  MoveL 8647 to (-40.61, 49.48, 125.68) mm, rotated rx 180 ry 0 rz 180 deg; joints [-136.108, -46.338, -97.928, 49.844, 65.111, -26.51]
  MoveL 8648 to (-40.61, 49.48, 125.68) mm, rotated rx 180 ry 0 rz 180 deg; joints [-136.108, -46.338, -97.928, 49.844, 65.111, -26.51]
  Call Extruder(456.97214)
  MoveL 8649 to (-40.56, 49.18, 125.68) mm, rotated rx 180 ry 0 rz -180 deg; joints [-136.149, -46.327, -97.959, 49.797, 65.104, -26.477]
  MoveL 8650 to (-40.56, 49.18, 125.68) mm, rotated rx 180 ry 0 rz -180 deg; joints [-136.149, -46.327, -97.959, 49.797, 65.104, -26.477]
  Call Extruder(457.10606)
  MoveL 8651 to (-40.52, 48.93, 125.68) mm, rotated rx 180 ry 0 rz 180 deg; joints [-136.184, -46.317, -97.983, 49.757, 65.098, -26.45]
  MoveL 8652 to (-40.52, 48.93, 125.68) mm, rotated rx 180 ry 0 rz 180 deg; joints [-136.184, -46.317, -97.983, 49.757, 65.098, -26.45]
  Call Extruder(457.24060)
  MoveL 8653 to (-40.47, 48.68, 125.68) mm, rotated rx 180 ry 0 rz -180 deg; joints [-136.219, -46.308, -98.006, 49.717, 65.092, -26.424]
  MoveL 8654 to (-40.47, 48.68, 125.68) mm, rotated rx 180 ry 0 rz -180 deg; joints [-136.219, -46.308, -98.006, 49.717, 65.092, -26.424]
  Call Extruder(457.37574)
  MoveL 8655 to (-40.42, 48.43, 125.68) mm, rotated rx 180 ry 0 rz 180 deg; joints [-136.254, -46.3, -98.03, 49.678, 65.086, -26.397]
  MoveL 8656 to (-40.42, 48.43, 125.68) mm, rotated rx 180 ry 0 rz 180 deg; joints [-136.254, -46.3, -98.03, 49.678, 65.086, -26.397]
  Call Extruder(457.51150)
  MoveL 8657 to (-40.37, 48.18, 125.68) mm, rotated rx 180 ry 0 rz 180 deg; joints [-136.288, -46.291, -98.053, 49.638, 65.08, -26.37]
  MoveL 8658 to (-40.37, 48.18, 125.68) mm, rotated rx 180 ry 0 rz 180 deg; joints [-136.288, -46.291, -98.053, 49.638, 65.08, -26.37]
  Call Extruder(457.64786)
  MoveL 8659 to (-40.32, 47.93, 125.68) mm, rotated rx 180 ry 0 rz 180 deg; joints [-136.323, -46.282, -98.077, 49.599, 65.074, -26.344]
  MoveL 8660 to (-40.32, 47.93, 125.68) mm, rotated rx 180 ry 0 rz 180 deg; joints [-136.323, -46.282, -98.077, 49.599, 65.074, -26.344]
  Call Extruder(457.78484)
  MoveL 8661 to (-40.27, 47.68, 125.68) mm, rotated rx 180 ry 0 rz 180 deg; joints [-136.358, -46.273, -98.1, 49.559, 65.068, -26.317]
  MoveL 8662 to (-40.27, 47.68, 125.68) mm, rotated rx 180 ry 0 rz 180 deg; joints [-136.358, -46.273, -98.1, 49.559, 65.068, -26.317]
  Call Extruder(457.92243)
  MoveL 8663 to (-40.22, 47.43, 125.68) mm, rotated rx 180 ry 0 rz 180 deg; joints [-136.393, -46.264, -98.123, 49.519, 65.062, -26.29]
  MoveL 8664 to (-40.22, 47.43, 125.68) mm, rotated rx 180 ry 0 rz 180 deg; joints [-136.393, -46.264, -98.123, 49.519, 65.062, -26.29]
  Call Extruder(458.03615)
  MoveL 8665 to (-40.17, 47.23, 125.68) mm, rotated rx -180 ry 0 rz -180 deg; joints [-136.422, -46.257, -98.142, 49.486, 65.056, -26.268]
  MoveL 8666 to (-40.17, 47.23, 125.68) mm, rotated rx -180 ry 0 rz -180 deg; joints [-136.422, -46.257, -98.142, 49.486, 65.056, -26.268]
  Call Extruder(458.15034)
  MoveL 8667 to (-40.13, 47.02, 125.68) mm, rotated rx 180 ry 0 rz 180 deg; joints [-136.452, -46.249, -98.161, 49.453, 65.051, -26.246]
  MoveL 8668 to (-40.13, 47.02, 125.68) mm, rotated rx 180 ry 0 rz 180 deg; joints [-136.452, -46.249, -98.161, 49.453, 65.051, -26.246]
  Call Extruder(458.26497)
  MoveL 8669 to (-40.08, 46.82, 125.68) mm, rotated rx 180 ry 0 rz 180 deg; joints [-136.481, -46.242, -98.18, 49.42, 65.046, -26.224]
  MoveL 8670 to (-40.08, 46.82, 125.68) mm, rotated rx 180 ry 0 rz 180 deg; joints [-136.481, -46.242, -98.18, 49.42, 65.046, -26.224]
  Call Extruder(458.38006)
  MoveL 8671 to (-40.04, 46.61, 125.68) mm, rotated rx 180 ry 0 rz -180 deg; joints [-136.51, -46.235, -98.198, 49.387, 65.04, -26.203]
  MoveL 8672 to (-40.04, 46.61, 125.68) mm, rotated rx 180 ry 0 rz -180 deg; joints [-136.51, -46.235, -98.198, 49.387, 65.04, -26.203]
  Call Extruder(458.50230)
  MoveL 8673 to (-39.98, 46.4, 125.68) mm, rotated rx 180 ry 0 rz -180 deg; joints [-136.542, -46.228, -98.217, 49.352, 65.034, -26.18]
  MoveL 8674 to (-39.98, 46.4, 125.68) mm, rotated rx 180 ry 0 rz -180 deg; joints [-136.542, -46.228, -98.217, 49.352, 65.034, -26.18]
  Call Extruder(458.63196)
  MoveL 8675 to (-39.92, 46.18, 125.68) mm, rotated rx 180 ry 0 rz -180 deg; joints [-136.576, -46.221, -98.235, 49.314, 65.026, -26.156]
  MoveL 8676 to (-39.92, 46.18, 125.68) mm, rotated rx 180 ry 0 rz -180 deg; joints [-136.576, -46.221, -98.235, 49.314, 65.026, -26.156]
  Call Extruder(458.76219)
  MoveL 8677 to (-39.85, 45.95, 125.68) mm, rotated rx -180 ry 0 rz -180 deg; joints [-136.61, -46.214, -98.253, 49.277, 65.018, -26.133]
  MoveL 8678 to (-39.85, 45.95, 125.68) mm, rotated rx -180 ry 0 rz -180 deg; joints [-136.61, -46.214, -98.253, 49.277, 65.018, -26.133]
  Call Extruder(458.89299)
  MoveL 8679 to (-39.78, 45.73, 125.68) mm, rotated rx -180 ry 0 rz 180 deg; joints [-136.644, -46.208, -98.271, 49.239, 65.01, -26.109]
  MoveL 8680 to (-39.78, 45.73, 125.68) mm, rotated rx -180 ry 0 rz 180 deg; joints [-136.644, -46.208, -98.271, 49.239, 65.01, -26.109]
  Call Extruder(459.02435)
  MoveL 8681 to (-39.71, 45.51, 125.68) mm, rotated rx 180 ry 0 rz 180 deg; joints [-136.678, -46.201, -98.289, 49.201, 65.002, -26.085]
  MoveL 8682 to (-39.71, 45.51, 125.68) mm, rotated rx 180 ry 0 rz 180 deg; joints [-136.678, -46.201, -98.289, 49.201, 65.002, -26.085]
  Call Extruder(459.13625)
  MoveL 8683 to (-39.65, 45.32, 125.68) mm, rotated rx 180 ry 0 rz -180 deg; joints [-136.707, -46.195, -98.303, 49.169, 64.996, -26.066]
  MoveL 8684 to (-39.65, 45.32, 125.68) mm, rotated rx 180 ry 0 rz -180 deg; joints [-136.707, -46.195, -98.303, 49.169, 64.996, -26.066]
  Call Extruder(459.24859)
  MoveL 8685 to (-39.59, 45.13, 125.68) mm, rotated rx -180 ry 0 rz 180 deg; joints [-136.737, -46.19, -98.318, 49.137, 64.989, -26.046]
  MoveL 8686 to (-39.59, 45.13, 125.68) mm, rotated rx -180 ry 0 rz 180 deg; joints [-136.737, -46.19, -98.318, 49.137, 64.989, -26.046]
  Call Extruder(459.36138)
  MoveL 8687 to (-39.53, 44.94, 125.68) mm, rotated rx 180 ry 0 rz 180 deg; joints [-136.766, -46.184, -98.332, 49.104, 64.982, -26.026]
  MoveL 8688 to (-39.53, 44.94, 125.68) mm, rotated rx 180 ry 0 rz 180 deg; joints [-136.766, -46.184, -98.332, 49.104, 64.982, -26.026]
  Call Extruder(459.47461)
  MoveL 8689 to (-39.47, 44.75, 125.68) mm, rotated rx 180 ry 0 rz -180 deg; joints [-136.796, -46.179, -98.347, 49.072, 64.975, -26.006]
  MoveL 8690 to (-39.47, 44.75, 125.68) mm, rotated rx 180 ry 0 rz -180 deg; joints [-136.796, -46.179, -98.347, 49.072, 64.975, -26.006]
  Call Extruder(459.58829)
  MoveL 8691 to (-39.41, 44.56, 125.68) mm, rotated rx -180 ry 0 rz 180 deg; joints [-136.825, -46.173, -98.361, 49.04, 64.968, -25.986]
  MoveL 8692 to (-39.41, 44.56, 125.68) mm, rotated rx -180 ry 0 rz 180 deg; joints [-136.825, -46.173, -98.361, 49.04, 64.968, -25.986]
  Call Extruder(459.77026)
  MoveL 8693 to (-39.29, 44.27, 125.68) mm, rotated rx 180 ry 0 rz -180 deg; joints [-136.873, -46.166, -98.381, 48.988, 64.954, -25.956]
  MoveL 8694 to (-39.29, 44.27, 125.68) mm, rotated rx 180 ry 0 rz -180 deg; joints [-136.873, -46.166, -98.381, 48.988, 64.954, -25.956]
  Call Extruder(459.95298)
  MoveL 8695 to (-39.17, 43.98, 125.68) mm, rotated rx 180 ry 0 rz -180 deg; joints [-136.922, -46.158, -98.4, 48.935, 64.941, -25.926]
  MoveL 8696 to (-39.17, 43.98, 125.68) mm, rotated rx 180 ry 0 rz -180 deg; joints [-136.922, -46.158, -98.4, 48.935, 64.941, -25.926]
  Call Extruder(460.12339)
  MoveL 8697 to (-39.05, 43.71, 125.68) mm, rotated rx 180 ry 0 rz 180 deg; joints [-136.967, -46.152, -98.417, 48.887, 64.928, -25.898]
  MoveL 8698 to (-39.05, 43.71, 125.68) mm, rotated rx 180 ry 0 rz 180 deg; joints [-136.967, -46.152, -98.417, 48.887, 64.928, -25.898]
  Call Extruder(460.28137)
  MoveL 8699 to (-38.94, 43.46, 125.68) mm, rotated rx 180 ry 0 rz 180 deg; joints [-137.009, -46.146, -98.433, 48.842, 64.916, -25.872]
  MoveL 8700 to (-38.94, 43.46, 125.68) mm, rotated rx 180 ry 0 rz 180 deg; joints [-137.009, -46.146, -98.433, 48.842, 64.916, -25.872]
  Call Extruder(460.43996)
  MoveL 8701 to (-38.84, 43.21, 125.68) mm, rotated rx -180 ry 0 rz 180 deg; joints [-137.05, -46.14, -98.449, 48.797, 64.905, -25.846]
  MoveL 8702 to (-38.84, 43.21, 125.68) mm, rotated rx -180 ry 0 rz 180 deg; joints [-137.05, -46.14, -98.449, 48.797, 64.905, -25.846]
  Call Extruder(460.64612)
  MoveL 8703 to (-38.66, 42.91, 125.68) mm, rotated rx -180 ry 0 rz -180 deg; joints [-137.107, -46.135, -98.462, 48.738, 64.886, -25.816]
  MoveL 8704 to (-38.66, 42.91, 125.68) mm, rotated rx -180 ry 0 rz -180 deg; joints [-137.107, -46.135, -98.462, 48.738, 64.886, -25.816]
  Call Extruder(460.85306)
  MoveL 8705 to (-38.49, 42.6, 125.68) mm, rotated rx -180 ry 0 rz -180 deg; joints [-137.163, -46.13, -98.476, 48.679, 64.867, -25.785]
  MoveL 8706 to (-38.49, 42.6, 125.68) mm, rotated rx -180 ry 0 rz -180 deg; joints [-137.163, -46.13, -98.476, 48.679, 64.867, -25.785]
  Call Extruder(461.06079)
  MoveL 8707 to (-38.31, 42.3, 125.68) mm, rotated rx 180 ry 0 rz 180 deg; joints [-137.219, -46.125, -98.489, 48.62, 64.848, -25.755]
  MoveL 8708 to (-38.31, 42.3, 125.68) mm, rotated rx 180 ry 0 rz 180 deg; joints [-137.219, -46.125, -98.489, 48.62, 64.848, -25.755]
  Call Extruder(461.26929)
  MoveL 8709 to (-38.13, 41.99, 125.68) mm, rotated rx 180 ry 0 rz -180 deg; joints [-137.275, -46.119, -98.502, 48.562, 64.829, -25.724]
  MoveL 8710 to (-38.13, 41.99, 125.68) mm, rotated rx 180 ry 0 rz -180 deg; joints [-137.275, -46.119, -98.502, 48.562, 64.829, -25.724]
  Call Extruder(461.44884)
  MoveL 8711 to (-37.96, 41.75, 125.68) mm, rotated rx 180 ry 0 rz 180 deg; joints [-137.324, -46.117, -98.509, 48.511, 64.81, -25.7]
  MoveL 8712 to (-37.96, 41.75, 125.68) mm, rotated rx 180 ry 0 rz 180 deg; joints [-137.324, -46.117, -98.509, 48.511, 64.81, -25.7]
  Call Extruder(461.78228)
  MoveL 8713 to (-37.63, 41.3, 125.68) mm, rotated rx 180 ry 0 rz -180 deg; joints [-137.415, -46.113, -98.52, 48.418, 64.775, -25.656]
  MoveL 8714 to (-37.63, 41.3, 125.68) mm, rotated rx 180 ry 0 rz -180 deg; joints [-137.415, -46.113, -98.52, 48.418, 64.775, -25.656]
  Call Extruder(462.11690)
  MoveL 8715 to (-37.3, 40.85, 125.68) mm, rotated rx 180 ry 0 rz 180 deg; joints [-137.506, -46.109, -98.531, 48.325, 64.74, -25.611]
  Call Extruder(462.94483)
  MoveL 8716 to (-36.39, 39.81, 125.68) mm, rotated rx 180 ry 0 rz -180 deg; joints [-137.733, -46.107, -98.535, 48.098, 64.644, -25.512]
  Call Extruder(463.77274)
  MoveL 8717 to (-35.35, 38.9, 125.68) mm, rotated rx 180 ry 0 rz -180 deg; joints [-137.958, -46.117, -98.508, 47.879, 64.536, -25.43]
  Call Extruder(463.94004)
  MoveL 8718 to (-35.13, 38.73, 125.68) mm, rotated rx 180 ry 0 rz 180 deg; joints [-138.003, -46.121, -98.498, 47.836, 64.513, -25.415]
  MoveL 8719 to (-35.13, 38.73, 125.68) mm, rotated rx 180 ry 0 rz 180 deg; joints [-138.003, -46.121, -98.498, 47.836, 64.513, -25.415]
  Call Extruder(464.27347)
  MoveL 8720 to (-34.68, 38.4, 125.68) mm, rotated rx -180 ry 0 rz 180 deg; joints [-138.092, -46.129, -98.478, 47.751, 64.466, -25.387]
  MoveL 8721 to (-34.68, 38.4, 125.68) mm, rotated rx -180 ry 0 rz 180 deg; joints [-138.092, -46.129, -98.478, 47.751, 64.466, -25.387]
  Call Extruder(464.60571)
  MoveL 8722 to (-34.23, 38.08, 125.68) mm, rotated rx -180 ry 0 rz -180 deg; joints [-138.182, -46.136, -98.458, 47.666, 64.419, -25.358]
  MoveL 8723 to (-34.23, 38.08, 125.68) mm, rotated rx -180 ry 0 rz -180 deg; joints [-138.182, -46.136, -98.458, 47.666, 64.419, -25.358]
  Call Extruder(464.72342)
  MoveL 8724 to (-34.05, 37.98, 125.68) mm, rotated rx 180 ry 0 rz -180 deg; joints [-138.213, -46.14, -98.447, 47.637, 64.402, -25.351]
  MoveL 8725 to (-34.05, 37.98, 125.68) mm, rotated rx 180 ry 0 rz -180 deg; joints [-138.213, -46.14, -98.447, 47.637, 64.402, -25.351]
  Call Extruder(464.93114)
  MoveL 8726 to (-33.75, 37.8, 125.68) mm, rotated rx 180 ry 0 rz 180 deg; joints [-138.267, -46.147, -98.429, 47.586, 64.371, -25.336]
  MoveL 8727 to (-33.75, 37.8, 125.68) mm, rotated rx 180 ry 0 rz 180 deg; joints [-138.267, -46.147, -98.429, 47.586, 64.371, -25.336]
  Call Extruder(465.13808)
  MoveL 8728 to (-33.45, 37.63, 125.68) mm, rotated rx -180 ry 0 rz 180 deg; joints [-138.322, -46.155, -98.41, 47.536, 64.339, -25.322]
  MoveL 8729 to (-33.45, 37.63, 125.68) mm, rotated rx -180 ry 0 rz 180 deg; joints [-138.322, -46.155, -98.41, 47.536, 64.339, -25.322]
  Call Extruder(465.34424)
  MoveL 8730 to (-33.14, 37.45, 125.68) mm, rotated rx 180 ry 0 rz -180 deg; joints [-138.376, -46.162, -98.39, 47.485, 64.308, -25.308]
  MoveL 8731 to (-33.14, 37.45, 125.68) mm, rotated rx 180 ry 0 rz -180 deg; joints [-138.376, -46.162, -98.39, 47.485, 64.308, -25.308]
  Call Extruder(465.52591)
  MoveL 8732 to (-32.87, 37.31, 125.68) mm, rotated rx -180 ry 0 rz -180 deg; joints [-138.424, -46.169, -98.371, 47.442, 64.28, -25.298]
  MoveL 8733 to (-32.87, 37.31, 125.68) mm, rotated rx -180 ry 0 rz -180 deg; joints [-138.424, -46.169, -98.371, 47.442, 64.28, -25.298]
  Call Extruder(465.68390)
  MoveL 8734 to (-32.62, 37.2, 125.68) mm, rotated rx 180 ry 0 rz -180 deg; joints [-138.464, -46.177, -98.351, 47.406, 64.254, -25.29]
  MoveL 8735 to (-32.62, 37.2, 125.68) mm, rotated rx 180 ry 0 rz -180 deg; joints [-138.464, -46.177, -98.351, 47.406, 64.254, -25.29]
  Call Extruder(465.84129)
  MoveL 8736 to (-32.37, 37.09, 125.68) mm, rotated rx -180 ry 0 rz -180 deg; joints [-138.504, -46.184, -98.331, 47.37, 64.229, -25.283]
  MoveL 8737 to (-32.37, 37.09, 125.68) mm, rotated rx -180 ry 0 rz -180 deg; joints [-138.504, -46.184, -98.331, 47.37, 64.229, -25.283]
  Call Extruder(465.98171)
  MoveL 8738 to (-32.14, 37, 125.68) mm, rotated rx -180 ry 0 rz -180 deg; joints [-138.54, -46.191, -98.313, 47.339, 64.206, -25.276]
  MoveL 8739 to (-32.14, 37, 125.68) mm, rotated rx -180 ry 0 rz -180 deg; joints [-138.54, -46.191, -98.313, 47.339, 64.206, -25.276]
  Call Extruder(466.13359)
  MoveL 8740 to (-31.9, 36.9, 125.68) mm, rotated rx -180 ry 0 rz 180 deg; joints [-138.579, -46.199, -98.293, 47.304, 64.181, -25.27]
  MoveL 8741 to (-31.9, 36.9, 125.68) mm, rotated rx -180 ry 0 rz 180 deg; joints [-138.579, -46.199, -98.293, 47.304, 64.181, -25.27]
  Call Extruder(466.29670)
  MoveL 8742 to (-31.64, 36.79, 125.68) mm, rotated rx 180 ry 0 rz 180 deg; joints [-138.62, -46.207, -98.271, 47.267, 64.154, -25.262]
  MoveL 8743 to (-31.64, 36.79, 125.68) mm, rotated rx 180 ry 0 rz 180 deg; joints [-138.62, -46.207, -98.271, 47.267, 64.154, -25.262]
  Call Extruder(466.41015)
  MoveL 8744 to (-31.45, 36.73, 125.68) mm, rotated rx 180 ry 0 rz 180 deg; joints [-138.648, -46.214, -98.254, 47.243, 64.135, -25.259]
  MoveL 8745 to (-31.45, 36.73, 125.68) mm, rotated rx 180 ry 0 rz 180 deg; joints [-138.648, -46.214, -98.254, 47.243, 64.135, -25.259]
  Call Extruder(466.52317)
  MoveL 8746 to (-31.26, 36.67, 125.68) mm, rotated rx 180 ry 0 rz 180 deg; joints [-138.676, -46.221, -98.237, 47.219, 64.116, -25.255]
  MoveL 8747 to (-31.26, 36.67, 125.68) mm, rotated rx 180 ry 0 rz 180 deg; joints [-138.676, -46.221, -98.237, 47.219, 64.116, -25.255]
  Call Extruder(466.63573)
  MoveL 8748 to (-31.07, 36.61, 125.68) mm, rotated rx 180 ry 0 rz 180 deg; joints [-138.704, -46.227, -98.219, 47.194, 64.096, -25.252]
  MoveL 8749 to (-31.07, 36.61, 125.68) mm, rotated rx 180 ry 0 rz 180 deg; joints [-138.704, -46.227, -98.219, 47.194, 64.096, -25.252]
  Call Extruder(466.74786)
  MoveL 8750 to (-30.88, 36.55, 125.68) mm, rotated rx -180 ry 0 rz 180 deg; joints [-138.732, -46.234, -98.202, 47.17, 64.077, -25.248]
  MoveL 8751 to (-30.88, 36.55, 125.68) mm, rotated rx -180 ry 0 rz 180 deg; joints [-138.732, -46.234, -98.202, 47.17, 64.077, -25.248]
  Call Extruder(466.85954)
  MoveL 8752 to (-30.7, 36.49, 125.68) mm, rotated rx -180 ry 0 rz -180 deg; joints [-138.759, -46.24, -98.184, 47.146, 64.058, -25.245]
  MoveL 8753 to (-30.7, 36.49, 125.68) mm, rotated rx -180 ry 0 rz -180 deg; joints [-138.759, -46.24, -98.184, 47.146, 64.058, -25.245]
  Call Extruder(466.99061)
  MoveL 8754 to (-30.47, 36.42, 125.68) mm, rotated rx 180 ry 0 rz 180 deg; joints [-138.792, -46.249, -98.163, 47.118, 64.035, -25.242]
  MoveL 8755 to (-30.47, 36.42, 125.68) mm, rotated rx 180 ry 0 rz 180 deg; joints [-138.792, -46.249, -98.163, 47.118, 64.035, -25.242]
  Call Extruder(467.12112)
  MoveL 8756 to (-30.25, 36.35, 125.68) mm, rotated rx 180 ry 0 rz 180 deg; joints [-138.824, -46.257, -98.142, 47.09, 64.012, -25.238]
  MoveL 8757 to (-30.25, 36.35, 125.68) mm, rotated rx 180 ry 0 rz 180 deg; joints [-138.824, -46.257, -98.142, 47.09, 64.012, -25.238]
  Call Extruder(467.25107)
  MoveL 8758 to (-30.02, 36.28, 125.68) mm, rotated rx 180 ry 0 rz -180 deg; joints [-138.856, -46.265, -98.12, 47.063, 63.99, -25.235]
  MoveL 8759 to (-30.02, 36.28, 125.68) mm, rotated rx 180 ry 0 rz -180 deg; joints [-138.856, -46.265, -98.12, 47.063, 63.99, -25.235]
  Call Extruder(467.38045)
  MoveL 8760 to (-29.8, 36.22, 125.68) mm, rotated rx 180 ry 0 rz -180 deg; joints [-138.889, -46.273, -98.099, 47.035, 63.967, -25.231]
  MoveL 8761 to (-29.8, 36.22, 125.68) mm, rotated rx 180 ry 0 rz -180 deg; joints [-138.889, -46.273, -98.099, 47.035, 63.967, -25.231]
  Call Extruder(467.50241)
  MoveL 8762 to (-29.59, 36.16, 125.68) mm, rotated rx 180 ry 0 rz 180 deg; joints [-138.919, -46.281, -98.078, 47.01, 63.945, -25.229]
  MoveL 8763 to (-29.59, 36.16, 125.68) mm, rotated rx 180 ry 0 rz 180 deg; joints [-138.919, -46.281, -98.078, 47.01, 63.945, -25.229]
  Call Extruder(467.61726)
  MoveL 8764 to (-29.38, 36.12, 125.68) mm, rotated rx -180 ry 0 rz -180 deg; joints [-138.946, -46.289, -98.056, 46.987, 63.924, -25.227]
  MoveL 8765 to (-29.38, 36.12, 125.68) mm, rotated rx -180 ry 0 rz -180 deg; joints [-138.946, -46.289, -98.056, 46.987, 63.924, -25.227]
  Call Extruder(467.73165)
  MoveL 8766 to (-29.18, 36.07, 125.68) mm, rotated rx 180 ry 0 rz 180 deg; joints [-138.973, -46.298, -98.035, 46.964, 63.904, -25.226]
  MoveL 8767 to (-29.18, 36.07, 125.68) mm, rotated rx 180 ry 0 rz 180 deg; joints [-138.973, -46.298, -98.035, 46.964, 63.904, -25.226]
  Call Extruder(467.84560)
  MoveL 8768 to (-28.97, 36.03, 125.68) mm, rotated rx 180 ry 0 rz -180 deg; joints [-139, -46.306, -98.013, 46.941, 63.883, -25.225]
  MoveL 8769 to (-28.97, 36.03, 125.68) mm, rotated rx 180 ry 0 rz -180 deg; joints [-139, -46.306, -98.013, 46.941, 63.883, -25.225]
  Call Extruder(467.95909)
  MoveL 8770 to (-28.77, 35.98, 125.68) mm, rotated rx 180 ry 0 rz -180 deg; joints [-139.028, -46.314, -97.991, 46.919, 63.862, -25.224]
  MoveL 8771 to (-28.77, 35.98, 125.68) mm, rotated rx 180 ry 0 rz -180 deg; joints [-139.028, -46.314, -97.991, 46.919, 63.862, -25.224]
  Call Extruder(468.09637)
  MoveL 8772 to (-28.52, 35.93, 125.68) mm, rotated rx -180 ry 0 rz -180 deg; joints [-139.06, -46.324, -97.965, 46.892, 63.837, -25.223]
  MoveL 8773 to (-28.52, 35.93, 125.68) mm, rotated rx -180 ry 0 rz -180 deg; joints [-139.06, -46.324, -97.965, 46.892, 63.837, -25.223]
  Call Extruder(468.23304)
  MoveL 8774 to (-28.27, 35.88, 125.68) mm, rotated rx 180 ry 0 rz 180 deg; joints [-139.093, -46.335, -97.938, 46.865, 63.812, -25.222]
  MoveL 8775 to (-28.27, 35.88, 125.68) mm, rotated rx 180 ry 0 rz 180 deg; joints [-139.093, -46.335, -97.938, 46.865, 63.812, -25.222]
  Call Extruder(468.36910)
  MoveL 8776 to (-28.02, 35.83, 125.68) mm, rotated rx 180 ry 0 rz -180 deg; joints [-139.126, -46.345, -97.911, 46.838, 63.786, -25.221]
  MoveL 8777 to (-28.02, 35.83, 125.68) mm, rotated rx 180 ry 0 rz -180 deg; joints [-139.126, -46.345, -97.911, 46.838, 63.786, -25.221]
  Call Extruder(468.50456)
  MoveL 8778 to (-27.77, 35.78, 125.68) mm, rotated rx 180 ry 0 rz 180 deg; joints [-139.158, -46.355, -97.884, 46.811, 63.761, -25.22]
  MoveL 8779 to (-27.77, 35.78, 125.68) mm, rotated rx 180 ry 0 rz 180 deg; joints [-139.158, -46.355, -97.884, 46.811, 63.761, -25.22]
  Call Extruder(468.63940)
  MoveL 8780 to (-27.52, 35.73, 125.68) mm, rotated rx 180 ry 0 rz 180 deg; joints [-139.191, -46.366, -97.857, 46.784, 63.736, -25.219]
  MoveL 8781 to (-27.52, 35.73, 125.68) mm, rotated rx 180 ry 0 rz 180 deg; joints [-139.191, -46.366, -97.857, 46.784, 63.736, -25.219]
  Call Extruder(468.77363)
  MoveL 8782 to (-27.28, 35.68, 125.68) mm, rotated rx -180 ry 0 rz 180 deg; joints [-139.223, -46.376, -97.83, 46.757, 63.711, -25.218]
  MoveL 8783 to (-27.28, 35.68, 125.68) mm, rotated rx -180 ry 0 rz 180 deg; joints [-139.223, -46.376, -97.83, 46.757, 63.711, -25.218]
  Call Extruder(468.90725)
  MoveL 8784 to (-27.03, 35.63, 125.68) mm, rotated rx -180 ry 0 rz 180 deg; joints [-139.256, -46.386, -97.803, 46.731, 63.686, -25.217]
  MoveL 8785 to (-27.03, 35.63, 125.68) mm, rotated rx -180 ry 0 rz 180 deg; joints [-139.256, -46.386, -97.803, 46.731, 63.686, -25.217]
  Call Extruder(469.06935)
  MoveL 8786 to (-26.72, 35.59, 125.68) mm, rotated rx -180 ry 0 rz 180 deg; joints [-139.294, -46.399, -97.768, 46.7, 63.655, -25.217]
  MoveL 8787 to (-26.72, 35.59, 125.68) mm, rotated rx -180 ry 0 rz 180 deg; joints [-139.294, -46.399, -97.768, 46.7, 63.655, -25.217]
  Call Extruder(469.23072)
  MoveL 8788 to (-26.41, 35.54, 125.68) mm, rotated rx 180 ry 0 rz 180 deg; joints [-139.332, -46.413, -97.734, 46.669, 63.624, -25.217]
  MoveL 8789 to (-26.41, 35.54, 125.68) mm, rotated rx 180 ry 0 rz 180 deg; joints [-139.332, -46.413, -97.734, 46.669, 63.624, -25.217]
  Call Extruder(469.39136)
  MoveL 8790 to (-26.11, 35.49, 125.68) mm, rotated rx 180 ry 0 rz -180 deg; joints [-139.371, -46.426, -97.699, 46.638, 63.593, -25.217]
  MoveL 8791 to (-26.11, 35.49, 125.68) mm, rotated rx 180 ry 0 rz -180 deg; joints [-139.371, -46.426, -97.699, 46.638, 63.593, -25.217]
  Call Extruder(469.55127)
  MoveL 8792 to (-25.8, 35.44, 125.68) mm, rotated rx 180 ry 0 rz -180 deg; joints [-139.409, -46.439, -97.664, 46.607, 63.562, -25.217]
  MoveL 8793 to (-25.8, 35.44, 125.68) mm, rotated rx 180 ry 0 rz -180 deg; joints [-139.409, -46.439, -97.664, 46.607, 63.562, -25.217]
  Call Extruder(469.71046)
  MoveL 8794 to (-25.5, 35.39, 125.68) mm, rotated rx 180 ry 0 rz -180 deg; joints [-139.447, -46.453, -97.63, 46.576, 63.531, -25.218]
  MoveL 8795 to (-25.5, 35.39, 125.68) mm, rotated rx 180 ry 0 rz -180 deg; joints [-139.447, -46.453, -97.63, 46.576, 63.531, -25.218]
  Call Extruder(469.86892)
  MoveL 8796 to (-25.19, 35.34, 125.68) mm, rotated rx 180 ry 0 rz 180 deg; joints [-139.485, -46.466, -97.595, 46.545, 63.5, -25.218]
  MoveL 8797 to (-25.19, 35.34, 125.68) mm, rotated rx 180 ry 0 rz 180 deg; joints [-139.485, -46.466, -97.595, 46.545, 63.5, -25.218]
  Call Extruder(470.06779)
  MoveL 8798 to (-24.8, 35.3, 125.68) mm, rotated rx -180 ry 0 rz 180 deg; joints [-139.531, -46.484, -97.549, 46.509, 63.461, -25.22]
  MoveL 8799 to (-24.8, 35.3, 125.68) mm, rotated rx -180 ry 0 rz 180 deg; joints [-139.531, -46.484, -97.549, 46.509, 63.461, -25.22]
  Call Extruder(470.26580)
  MoveL 8800 to (-24.42, 35.25, 125.68) mm, rotated rx 180 ry 0 rz 180 deg; joints [-139.577, -46.501, -97.503, 46.472, 63.421, -25.222]
  MoveL 8801 to (-24.42, 35.25, 125.68) mm, rotated rx 180 ry 0 rz 180 deg; joints [-139.577, -46.501, -97.503, 46.472, 63.421, -25.222]
  Call Extruder(470.46294)
  MoveL 8802 to (-24.03, 35.21, 125.68) mm, rotated rx -180 ry 0 rz 180 deg; joints [-139.624, -46.519, -97.457, 46.436, 63.382, -25.224]
  MoveL 8803 to (-24.03, 35.21, 125.68) mm, rotated rx -180 ry 0 rz 180 deg; joints [-139.624, -46.519, -97.457, 46.436, 63.382, -25.224]
  Call Extruder(470.65922)
  MoveL 8804 to (-23.64, 35.16, 125.68) mm, rotated rx 180 ry 0 rz -180 deg; joints [-139.67, -46.537, -97.411, 46.399, 63.343, -25.226]
  MoveL 8805 to (-23.64, 35.16, 125.68) mm, rotated rx 180 ry 0 rz -180 deg; joints [-139.67, -46.537, -97.411, 46.399, 63.343, -25.226]
  Call Extruder(470.90490)
  MoveL 8806 to (-23.15, 35.11, 125.68) mm, rotated rx 180 ry 0 rz 180 deg; joints [-139.726, -46.559, -97.352, 46.356, 63.294, -25.23]
  MoveL 8807 to (-23.15, 35.11, 125.68) mm, rotated rx 180 ry 0 rz 180 deg; joints [-139.726, -46.559, -97.352, 46.356, 63.294, -25.23]
  Call Extruder(471.19963)
  MoveL 8808 to (-22.56, 35.07, 125.68) mm, rotated rx -180 ry 0 rz -180 deg; joints [-139.793, -46.587, -97.279, 46.304, 63.234, -25.236]
  MoveL 8809 to (-22.56, 35.07, 125.68) mm, rotated rx -180 ry 0 rz -180 deg; joints [-139.793, -46.587, -97.279, 46.304, 63.234, -25.236]
  Call Extruder(471.49303)
  MoveL 8810 to (-21.97, 35.02, 125.68) mm, rotated rx -180 ry 0 rz 180 deg; joints [-139.86, -46.616, -97.206, 46.253, 63.175, -25.241]
  MoveL 8811 to (-21.97, 35.02, 125.68) mm, rotated rx -180 ry 0 rz 180 deg; joints [-139.86, -46.616, -97.206, 46.253, 63.175, -25.241]
  Call Extruder(471.92636)
  MoveL 8812 to (-21.1, 34.97, 125.68) mm, rotated rx -180 ry 0 rz -180 deg; joints [-139.956, -46.658, -97.095, 46.18, 63.087, -25.253]
  MoveL 8813 to (-21.1, 34.97, 125.68) mm, rotated rx -180 ry 0 rz -180 deg; joints [-139.956, -46.658, -97.095, 46.18, 63.087, -25.253]
  Call Extruder(472.49852)
  MoveL 8814 to (-19.94, 34.93, 125.68) mm, rotated rx 180 ry 0 rz 180 deg; joints [-140.081, -46.716, -96.945, 46.087, 62.97, -25.269]
  MoveL 8815 to (-19.94, 34.93, 125.68) mm, rotated rx 180 ry 0 rz 180 deg; joints [-140.081, -46.716, -96.945, 46.087, 62.97, -25.269]
  Call Extruder(472.92635)
  MoveL 8816 to (-19.06, 34.91, 125.68) mm, rotated rx 180 ry 0 rz 180 deg; joints [-140.173, -46.761, -96.831, 46.02, 62.882, -25.284]
  Call Extruder(589.57504)
  MoveL 8817 to (219.06, 34.91, 125.68) mm, rotated rx 180 ry 0 rz -180 deg; joints [-155.896, -65.517, -54.51, 41.799, 37.786, -35.244]
  MoveL 8818 to (219.06, 34.91, 125.68) mm, rotated rx 180 ry 0 rz -180 deg; joints [-155.896, -65.517, -54.51, 41.799, 37.786, -35.244]
  Call Extruder(590.29061)
  MoveL 8819 to (220.52, 34.95, 125.68) mm, rotated rx -180 ry 0 rz 180 deg; joints [-155.953, -65.686, -54.157, 41.882, 37.617, -35.385]
  MoveL 8820 to (220.52, 34.95, 125.68) mm, rotated rx -180 ry 0 rz 180 deg; joints [-155.953, -65.686, -54.157, 41.882, 37.617, -35.385]
  Call Extruder(590.86535)
  MoveL 8821 to (221.68, 35, 125.68) mm, rotated rx 180 ry 0 rz 180 deg; joints [-155.997, -65.823, -53.872, 41.952, 37.481, -35.501]
  MoveL 8822 to (221.68, 35, 125.68) mm, rotated rx 180 ry 0 rz 180 deg; joints [-155.997, -65.823, -53.872, 41.952, 37.481, -35.501]
  Call Extruder(591.15874)
  MoveL 8823 to (222.27, 35.04, 125.68) mm, rotated rx 180 ry 0 rz 180 deg; joints [-156.017, -65.894, -53.724, 41.993, 37.412, -35.564]
  MoveL 8824 to (222.27, 35.04, 125.68) mm, rotated rx 180 ry 0 rz 180 deg; joints [-156.017, -65.894, -53.724, 41.993, 37.412, -35.564]
  Call Extruder(591.45347)
  MoveL 8825 to (222.86, 35.09, 125.68) mm, rotated rx 180 ry 0 rz -180 deg; joints [-156.037, -65.965, -53.577, 42.033, 37.344, -35.628]
  MoveL 8826 to (222.86, 35.09, 125.68) mm, rotated rx 180 ry 0 rz -180 deg; joints [-156.037, -65.965, -53.577, 42.033, 37.344, -35.628]
  Call Extruder(591.74952)
  MoveL 8827 to (223.45, 35.14, 125.68) mm, rotated rx -180 ry 0 rz 180 deg; joints [-156.057, -66.036, -53.428, 42.074, 37.275, -35.692]
  MoveL 8828 to (223.45, 35.14, 125.68) mm, rotated rx -180 ry 0 rz 180 deg; joints [-156.057, -66.036, -53.428, 42.074, 37.275, -35.692]
  Call Extruder(591.94580)
  MoveL 8829 to (223.83, 35.18, 125.68) mm, rotated rx 180 ry 0 rz 180 deg; joints [-156.068, -66.083, -53.329, 42.104, 37.23, -35.736]
  MoveL 8830 to (223.83, 35.18, 125.68) mm, rotated rx 180 ry 0 rz 180 deg; joints [-156.068, -66.083, -53.329, 42.104, 37.23, -35.736]
  Call Extruder(592.14294)
  MoveL 8831 to (224.22, 35.23, 125.68) mm, rotated rx 180 ry 0 rz 180 deg; joints [-156.08, -66.131, -53.23, 42.134, 37.185, -35.781]
  MoveL 8832 to (224.22, 35.23, 125.68) mm, rotated rx 180 ry 0 rz 180 deg; joints [-156.08, -66.131, -53.23, 42.134, 37.185, -35.781]
  Call Extruder(592.34095)
  MoveL 8833 to (224.61, 35.27, 125.68) mm, rotated rx -180 ry 0 rz 180 deg; joints [-156.092, -66.179, -53.13, 42.164, 37.14, -35.826]
  MoveL 8834 to (224.61, 35.27, 125.68) mm, rotated rx -180 ry 0 rz 180 deg; joints [-156.092, -66.179, -53.13, 42.164, 37.14, -35.826]
  Call Extruder(592.53982)
  MoveL 8835 to (225, 35.32, 125.68) mm, rotated rx 180 ry 0 rz -180 deg; joints [-156.103, -66.227, -53.031, 42.194, 37.094, -35.871]
  MoveL 8836 to (225, 35.32, 125.68) mm, rotated rx 180 ry 0 rz -180 deg; joints [-156.103, -66.227, -53.031, 42.194, 37.094, -35.871]
  Call Extruder(592.71890)
  MoveL 8837 to (225.34, 35.37, 125.68) mm, rotated rx 180 ry 0 rz -180 deg; joints [-156.113, -66.27, -52.941, 42.223, 37.054, -35.913]
  MoveL 8838 to (225.34, 35.37, 125.68) mm, rotated rx 180 ry 0 rz -180 deg; joints [-156.113, -66.27, -52.941, 42.223, 37.054, -35.913]
  Call Extruder(592.87809)
  MoveL 8839 to (225.65, 35.42, 125.68) mm, rotated rx 180 ry 0 rz 180 deg; joints [-156.121, -66.309, -52.861, 42.249, 37.019, -35.951]
  MoveL 8840 to (225.65, 35.42, 125.68) mm, rotated rx 180 ry 0 rz 180 deg; joints [-156.121, -66.309, -52.861, 42.249, 37.019, -35.951]
  Call Extruder(593.03800)
  MoveL 8841 to (225.96, 35.47, 125.68) mm, rotated rx 180 ry 0 rz -180 deg; joints [-156.129, -66.347, -52.78, 42.275, 36.983, -35.989]
  MoveL 8842 to (225.96, 35.47, 125.68) mm, rotated rx 180 ry 0 rz -180 deg; joints [-156.129, -66.347, -52.78, 42.275, 36.983, -35.989]
  Call Extruder(593.19864)
  MoveL 8843 to (226.26, 35.51, 125.68) mm, rotated rx 180 ry 0 rz 180 deg; joints [-156.137, -66.386, -52.7, 42.302, 36.948, -36.027]
  MoveL 8844 to (226.26, 35.51, 125.68) mm, rotated rx 180 ry 0 rz 180 deg; joints [-156.137, -66.386, -52.7, 42.302, 36.948, -36.027]
  Call Extruder(593.36001)
  MoveL 8845 to (226.57, 35.56, 125.68) mm, rotated rx -180 ry 0 rz -180 deg; joints [-156.145, -66.425, -52.62, 42.329, 36.912, -36.065]
  MoveL 8846 to (226.57, 35.56, 125.68) mm, rotated rx -180 ry 0 rz -180 deg; joints [-156.145, -66.425, -52.62, 42.329, 36.912, -36.065]
  Call Extruder(593.52210)
  MoveL 8847 to (226.87, 35.61, 125.68) mm, rotated rx -180 ry 0 rz 180 deg; joints [-156.153, -66.463, -52.539, 42.355, 36.877, -36.103]
  MoveL 8848 to (226.87, 35.61, 125.68) mm, rotated rx -180 ry 0 rz 180 deg; joints [-156.153, -66.463, -52.539, 42.355, 36.877, -36.103]
  Call Extruder(593.67030)
  MoveL 8849 to (227.15, 35.66, 125.68) mm, rotated rx -180 ry 0 rz 180 deg; joints [-156.16, -66.499, -52.466, 42.381, 36.844, -36.139]
  MoveL 8850 to (227.15, 35.66, 125.68) mm, rotated rx -180 ry 0 rz 180 deg; joints [-156.16, -66.499, -52.466, 42.381, 36.844, -36.139]
  Call Extruder(593.80453)
  MoveL 8851 to (227.4, 35.71, 125.68) mm, rotated rx 180 ry 0 rz 180 deg; joints [-156.165, -66.531, -52.399, 42.404, 36.816, -36.172]
  MoveL 8852 to (227.4, 35.71, 125.68) mm, rotated rx 180 ry 0 rz 180 deg; joints [-156.165, -66.531, -52.399, 42.404, 36.816, -36.172]
  Call Extruder(593.93938)
  MoveL 8853 to (227.65, 35.76, 125.68) mm, rotated rx 180 ry 0 rz 180 deg; joints [-156.171, -66.563, -52.332, 42.428, 36.787, -36.205]
  MoveL 8854 to (227.65, 35.76, 125.68) mm, rotated rx 180 ry 0 rz 180 deg; joints [-156.171, -66.563, -52.332, 42.428, 36.787, -36.205]
  Call Extruder(594.07483)
  MoveL 8855 to (227.9, 35.81, 125.68) mm, rotated rx -180 ry 0 rz 180 deg; joints [-156.176, -66.595, -52.265, 42.452, 36.758, -36.238]
  MoveL 8856 to (227.9, 35.81, 125.68) mm, rotated rx -180 ry 0 rz 180 deg; joints [-156.176, -66.595, -52.265, 42.452, 36.758, -36.238]
  Call Extruder(594.21089)
  MoveL 8857 to (228.15, 35.86, 125.68) mm, rotated rx -180 ry 0 rz 180 deg; joints [-156.182, -66.628, -52.198, 42.476, 36.729, -36.271]
  MoveL 8858 to (228.15, 35.86, 125.68) mm, rotated rx -180 ry 0 rz 180 deg; joints [-156.182, -66.628, -52.198, 42.476, 36.729, -36.271]
  Call Extruder(594.34757)
  MoveL 8859 to (228.4, 35.91, 125.68) mm, rotated rx 180 ry 0 rz 180 deg; joints [-156.187, -66.66, -52.131, 42.5, 36.7, -36.304]
  MoveL 8860 to (228.4, 35.91, 125.68) mm, rotated rx 180 ry 0 rz 180 deg; joints [-156.187, -66.66, -52.131, 42.5, 36.7, -36.304]
  Call Extruder(594.48485)
  MoveL 8861 to (228.64, 35.96, 125.68) mm, rotated rx 180 ry 0 rz 180 deg; joints [-156.193, -66.692, -52.064, 42.524, 36.671, -36.338]
  MoveL 8862 to (228.64, 35.96, 125.68) mm, rotated rx 180 ry 0 rz 180 deg; joints [-156.193, -66.692, -52.064, 42.524, 36.671, -36.338]
  Call Extruder(594.61052)
  MoveL 8863 to (228.87, 36, 125.68) mm, rotated rx 180 ry 0 rz 180 deg; joints [-156.198, -66.722, -52.002, 42.546, 36.645, -36.368]
  MoveL 8864 to (228.87, 36, 125.68) mm, rotated rx 180 ry 0 rz 180 deg; joints [-156.198, -66.722, -52.002, 42.546, 36.645, -36.368]
  Call Extruder(594.72447)
  MoveL 8865 to (229.08, 36.05, 125.68) mm, rotated rx 180 ry 0 rz 180 deg; joints [-156.202, -66.749, -51.947, 42.567, 36.621, -36.397]
  MoveL 8866 to (229.08, 36.05, 125.68) mm, rotated rx 180 ry 0 rz 180 deg; joints [-156.202, -66.749, -51.947, 42.567, 36.621, -36.397]
  Call Extruder(594.83887)
  MoveL 8867 to (229.28, 36.09, 125.68) mm, rotated rx 180 ry 0 rz -180 deg; joints [-156.206, -66.776, -51.891, 42.587, 36.597, -36.425]
  MoveL 8868 to (229.28, 36.09, 125.68) mm, rotated rx 180 ry 0 rz -180 deg; joints [-156.206, -66.776, -51.891, 42.587, 36.597, -36.425]
  Call Extruder(594.95372)
  MoveL 8869 to (229.48, 36.14, 125.68) mm, rotated rx -180 ry 0 rz 180 deg; joints [-156.21, -66.802, -51.835, 42.608, 36.574, -36.453]
  MoveL 8870 to (229.48, 36.14, 125.68) mm, rotated rx -180 ry 0 rz 180 deg; joints [-156.21, -66.802, -51.835, 42.608, 36.574, -36.453]
  Call Extruder(595.06902)
  MoveL 8871 to (229.69, 36.18, 125.68) mm, rotated rx 180 ry 0 rz -180 deg; joints [-156.214, -66.829, -51.78, 42.629, 36.55, -36.481]
  MoveL 8872 to (229.69, 36.18, 125.68) mm, rotated rx 180 ry 0 rz -180 deg; joints [-156.214, -66.829, -51.78, 42.629, 36.55, -36.481]
  Call Extruder(595.20041)
  MoveL 8873 to (229.92, 36.25, 125.68) mm, rotated rx -180 ry 0 rz -180 deg; joints [-156.218, -66.86, -51.716, 42.655, 36.524, -36.516]
  MoveL 8874 to (229.92, 36.25, 125.68) mm, rotated rx -180 ry 0 rz -180 deg; joints [-156.218, -66.86, -51.716, 42.655, 36.524, -36.516]
  Call Extruder(595.31352)
  MoveL 8875 to (230.11, 36.31, 125.68) mm, rotated rx 180 ry 0 rz 180 deg; joints [-156.22, -66.887, -51.661, 42.678, 36.501, -36.545]
  MoveL 8876 to (230.11, 36.31, 125.68) mm, rotated rx 180 ry 0 rz 180 deg; joints [-156.22, -66.887, -51.661, 42.678, 36.501, -36.545]
  Call Extruder(595.42707)
  MoveL 8877 to (230.31, 36.37, 125.68) mm, rotated rx 180 ry 0 rz 180 deg; joints [-156.222, -66.913, -51.605, 42.701, 36.479, -36.575]
  MoveL 8878 to (230.31, 36.37, 125.68) mm, rotated rx 180 ry 0 rz 180 deg; joints [-156.222, -66.913, -51.605, 42.701, 36.479, -36.575]
  Call Extruder(595.54106)
  MoveL 8879 to (230.5, 36.43, 125.68) mm, rotated rx -180 ry 0 rz 180 deg; joints [-156.225, -66.94, -51.55, 42.724, 36.456, -36.605]
  MoveL 8880 to (230.5, 36.43, 125.68) mm, rotated rx -180 ry 0 rz 180 deg; joints [-156.225, -66.94, -51.55, 42.724, 36.456, -36.605]
  Call Extruder(595.65549)
  MoveL 8881 to (230.69, 36.49, 125.68) mm, rotated rx 180 ry 0 rz 180 deg; joints [-156.227, -66.967, -51.495, 42.747, 36.434, -36.635]
  MoveL 8882 to (230.69, 36.49, 125.68) mm, rotated rx 180 ry 0 rz 180 deg; joints [-156.227, -66.967, -51.495, 42.747, 36.434, -36.635]
  Call Extruder(595.76739)
  MoveL 8883 to (230.88, 36.55, 125.68) mm, rotated rx 180 ry 0 rz 180 deg; joints [-156.229, -66.993, -51.441, 42.77, 36.412, -36.665]
  MoveL 8884 to (230.88, 36.55, 125.68) mm, rotated rx 180 ry 0 rz 180 deg; joints [-156.229, -66.993, -51.441, 42.77, 36.412, -36.665]
  Call Extruder(595.87973)
  MoveL 8885 to (231.07, 36.61, 125.68) mm, rotated rx 180 ry 0 rz 180 deg; joints [-156.231, -67.019, -51.387, 42.793, 36.391, -36.695]
  MoveL 8886 to (231.07, 36.61, 125.68) mm, rotated rx 180 ry 0 rz 180 deg; joints [-156.231, -67.019, -51.387, 42.793, 36.391, -36.695]
  Call Extruder(595.99252)
  MoveL 8887 to (231.26, 36.67, 125.68) mm, rotated rx -180 ry 0 rz 180 deg; joints [-156.233, -67.045, -51.333, 42.816, 36.369, -36.725]
  MoveL 8888 to (231.26, 36.67, 125.68) mm, rotated rx -180 ry 0 rz 180 deg; joints [-156.233, -67.045, -51.333, 42.816, 36.369, -36.725]
  Call Extruder(596.10575)
  MoveL 8889 to (231.45, 36.73, 125.68) mm, rotated rx -180 ry 0 rz 180 deg; joints [-156.235, -67.071, -51.279, 42.839, 36.347, -36.755]
  MoveL 8890 to (231.45, 36.73, 125.68) mm, rotated rx -180 ry 0 rz 180 deg; joints [-156.235, -67.071, -51.279, 42.839, 36.347, -36.755]
  Call Extruder(596.21943)
  MoveL 8891 to (231.64, 36.79, 125.68) mm, rotated rx 180 ry 0 rz 180 deg; joints [-156.237, -67.097, -51.225, 42.862, 36.326, -36.785]
  MoveL 8892 to (231.64, 36.79, 125.68) mm, rotated rx 180 ry 0 rz 180 deg; joints [-156.237, -67.097, -51.225, 42.862, 36.326, -36.785]
  Call Extruder(596.40139)
  MoveL 8893 to (231.93, 36.91, 125.68) mm, rotated rx -180 ry 0 rz 180 deg; joints [-156.238, -67.139, -51.139, 42.903, 36.292, -36.835]
  MoveL 8894 to (231.93, 36.91, 125.68) mm, rotated rx -180 ry 0 rz 180 deg; joints [-156.238, -67.139, -51.139, 42.903, 36.292, -36.835]
  Call Extruder(596.58411)
  MoveL 8895 to (232.22, 37.03, 125.68) mm, rotated rx -180 ry 0 rz 180 deg; joints [-156.238, -67.181, -51.052, 42.943, 36.259, -36.886]
  MoveL 8896 to (232.22, 37.03, 125.68) mm, rotated rx -180 ry 0 rz 180 deg; joints [-156.238, -67.181, -51.052, 42.943, 36.259, -36.886]
  Call Extruder(596.75452)
  MoveL 8897 to (232.49, 37.15, 125.68) mm, rotated rx 180 ry 0 rz 180 deg; joints [-156.239, -67.22, -50.971, 42.982, 36.228, -36.934]
  MoveL 8898 to (232.49, 37.15, 125.68) mm, rotated rx 180 ry 0 rz 180 deg; joints [-156.239, -67.22, -50.971, 42.982, 36.228, -36.934]
  Call Extruder(596.91252)
  MoveL 8899 to (232.74, 37.26, 125.68) mm, rotated rx -180 ry 0 rz 180 deg; joints [-156.239, -67.256, -50.897, 43.017, 36.2, -36.978]
  MoveL 8900 to (232.74, 37.26, 125.68) mm, rotated rx -180 ry 0 rz 180 deg; joints [-156.239, -67.256, -50.897, 43.017, 36.2, -36.978]
  Call Extruder(597.07112)
  MoveL 8901 to (232.99, 37.36, 125.68) mm, rotated rx -180 ry 0 rz -180 deg; joints [-156.239, -67.292, -50.822, 43.053, 36.172, -37.023]
  MoveL 8902 to (232.99, 37.36, 125.68) mm, rotated rx -180 ry 0 rz -180 deg; joints [-156.239, -67.292, -50.822, 43.053, 36.172, -37.023]
  Call Extruder(597.27729)
  MoveL 8903 to (233.29, 37.54, 125.68) mm, rotated rx -180 ry 0 rz 180 deg; joints [-156.236, -67.338, -50.725, 43.104, 36.137, -37.084]
  MoveL 8904 to (233.29, 37.54, 125.68) mm, rotated rx -180 ry 0 rz 180 deg; joints [-156.236, -67.338, -50.725, 43.104, 36.137, -37.084]
  Call Extruder(597.48423)
  MoveL 8905 to (233.6, 37.71, 125.68) mm, rotated rx -180 ry 0 rz 180 deg; joints [-156.232, -67.385, -50.629, 43.156, 36.103, -37.146]
  MoveL 8906 to (233.6, 37.71, 125.68) mm, rotated rx -180 ry 0 rz 180 deg; joints [-156.232, -67.385, -50.629, 43.156, 36.103, -37.146]
  Call Extruder(597.69196)
  MoveL 8907 to (233.9, 37.89, 125.68) mm, rotated rx 180 ry 0 rz 180 deg; joints [-156.228, -67.432, -50.532, 43.208, 36.069, -37.208]
  MoveL 8908 to (233.9, 37.89, 125.68) mm, rotated rx 180 ry 0 rz 180 deg; joints [-156.228, -67.432, -50.532, 43.208, 36.069, -37.208]
  Call Extruder(597.90046)
  MoveL 8909 to (234.21, 38.06, 125.68) mm, rotated rx 180 ry 0 rz 180 deg; joints [-156.224, -67.478, -50.436, 43.26, 36.035, -37.271]
  MoveL 8910 to (234.21, 38.06, 125.68) mm, rotated rx 180 ry 0 rz 180 deg; joints [-156.224, -67.478, -50.436, 43.26, 36.035, -37.271]
  Call Extruder(598.08001)
  MoveL 8911 to (234.45, 38.24, 125.68) mm, rotated rx 180 ry 0 rz 180 deg; joints [-156.218, -67.518, -50.354, 43.309, 36.008, -37.327]
  MoveL 8912 to (234.45, 38.24, 125.68) mm, rotated rx 180 ry 0 rz 180 deg; joints [-156.218, -67.518, -50.354, 43.309, 36.008, -37.327]
  Call Extruder(598.41342)
  MoveL 8913 to (234.9, 38.57, 125.68) mm, rotated rx 180 ry 0 rz -180 deg; joints [-156.206, -67.591, -50.202, 43.398, 35.958, -37.431]
  MoveL 8914 to (234.9, 38.57, 125.68) mm, rotated rx 180 ry 0 rz -180 deg; joints [-156.206, -67.591, -50.202, 43.398, 35.958, -37.431]
  Call Extruder(598.74802)
  MoveL 8915 to (235.35, 38.9, 125.68) mm, rotated rx 180 ry 0 rz 180 deg; joints [-156.195, -67.665, -50.05, 43.489, 35.908, -37.536]
  Call Extruder(599.57597)
  MoveL 8916 to (236.39, 39.81, 125.68) mm, rotated rx 180 ry 0 rz 180 deg; joints [-156.154, -67.843, -49.682, 43.725, 35.796, -37.804]
  Call Extruder(600.40391)
  MoveL 8917 to (237.3, 40.85, 125.68) mm, rotated rx -180 ry 0 rz 180 deg; joints [-156.097, -68.014, -49.329, 43.977, 35.7, -38.082]
  Call Extruder(600.57121)
  MoveL 8918 to (237.47, 41.07, 125.68) mm, rotated rx -180 ry 0 rz -180 deg; joints [-156.083, -68.047, -49.261, 44.03, 35.683, -38.139]
  MoveL 8919 to (237.47, 41.07, 125.68) mm, rotated rx -180 ry 0 rz -180 deg; joints [-156.083, -68.047, -49.261, 44.03, 35.683, -38.139]
  Call Extruder(600.90463)
  MoveL 8920 to (237.79, 41.52, 125.68) mm, rotated rx -180 ry 0 rz 180 deg; joints [-156.055, -68.113, -49.125, 44.135, 35.65, -38.253]
  MoveL 8921 to (237.79, 41.52, 125.68) mm, rotated rx -180 ry 0 rz 180 deg; joints [-156.055, -68.113, -49.125, 44.135, 35.65, -38.253]
  Call Extruder(601.23686)
  MoveL 8922 to (238.12, 41.98, 125.68) mm, rotated rx 180 ry 0 rz -180 deg; joints [-156.028, -68.18, -48.988, 44.241, 35.616, -38.367]
  MoveL 8923 to (238.12, 41.98, 125.68) mm, rotated rx 180 ry 0 rz -180 deg; joints [-156.028, -68.18, -48.988, 44.241, 35.616, -38.367]
  Call Extruder(601.35455)
  MoveL 8924 to (238.22, 42.15, 125.68) mm, rotated rx -180 ry 0 rz -180 deg; joints [-156.016, -68.202, -48.943, 44.279, 35.607, -38.408]
  MoveL 8925 to (238.22, 42.15, 125.68) mm, rotated rx -180 ry 0 rz -180 deg; joints [-156.016, -68.202, -48.943, 44.279, 35.607, -38.408]
  Call Extruder(601.56228)
  MoveL 8926 to (238.4, 42.45, 125.68) mm, rotated rx -180 ry 0 rz -180 deg; joints [-155.996, -68.241, -48.862, 44.346, 35.59, -38.48]
  MoveL 8927 to (238.4, 42.45, 125.68) mm, rotated rx -180 ry 0 rz -180 deg; joints [-155.996, -68.241, -48.862, 44.346, 35.59, -38.48]
  Call Extruder(601.76922)
  MoveL 8928 to (238.57, 42.75, 125.68) mm, rotated rx 180 ry 0 rz 180 deg; joints [-155.976, -68.28, -48.781, 44.414, 35.573, -38.552]
  MoveL 8929 to (238.57, 42.75, 125.68) mm, rotated rx 180 ry 0 rz 180 deg; joints [-155.976, -68.28, -48.781, 44.414, 35.573, -38.552]
  Call Extruder(601.97539)
  MoveL 8930 to (238.75, 43.06, 125.68) mm, rotated rx -180 ry 0 rz -180 deg; joints [-155.956, -68.319, -48.701, 44.482, 35.556, -38.624]
  MoveL 8931 to (238.75, 43.06, 125.68) mm, rotated rx -180 ry 0 rz -180 deg; joints [-155.956, -68.319, -48.701, 44.482, 35.556, -38.624]
  Call Extruder(602.15708)
  MoveL 8932 to (238.89, 43.33, 125.68) mm, rotated rx 180 ry 0 rz 180 deg; joints [-155.937, -68.352, -48.632, 44.543, 35.542, -38.688]
  MoveL 8933 to (238.89, 43.33, 125.68) mm, rotated rx 180 ry 0 rz 180 deg; joints [-155.937, -68.352, -48.632, 44.543, 35.542, -38.688]
  Call Extruder(602.31509)
  MoveL 8934 to (239, 43.58, 125.68) mm, rotated rx -180 ry 0 rz -180 deg; joints [-155.919, -68.38, -48.575, 44.596, 35.533, -38.743]
  MoveL 8935 to (239, 43.58, 125.68) mm, rotated rx -180 ry 0 rz -180 deg; joints [-155.919, -68.38, -48.575, 44.596, 35.533, -38.743]
  Call Extruder(602.47250)
  MoveL 8936 to (239.11, 43.83, 125.68) mm, rotated rx 180 ry 0 rz -180 deg; joints [-155.901, -68.408, -48.518, 44.648, 35.523, -38.798]
  MoveL 8937 to (239.11, 43.83, 125.68) mm, rotated rx 180 ry 0 rz -180 deg; joints [-155.901, -68.408, -48.518, 44.648, 35.523, -38.798]
  Call Extruder(602.65521)
  MoveL 8938 to (239.23, 44.12, 125.68) mm, rotated rx -180 ry 0 rz 180 deg; joints [-155.879, -68.439, -48.453, 44.71, 35.513, -38.862]
  MoveL 8939 to (239.23, 44.12, 125.68) mm, rotated rx -180 ry 0 rz 180 deg; joints [-155.879, -68.439, -48.453, 44.71, 35.513, -38.862]
  Call Extruder(602.83717)
  MoveL 8940 to (239.35, 44.42, 125.68) mm, rotated rx -180 ry 0 rz -180 deg; joints [-155.858, -68.471, -48.387, 44.772, 35.502, -38.926]
  MoveL 8941 to (239.35, 44.42, 125.68) mm, rotated rx -180 ry 0 rz -180 deg; joints [-155.858, -68.471, -48.387, 44.772, 35.502, -38.926]
  Call Extruder(602.98450)
  MoveL 8942 to (239.44, 44.66, 125.68) mm, rotated rx -180 ry 0 rz -180 deg; joints [-155.84, -68.496, -48.335, 44.822, 35.494, -38.977]
  MoveL 8943 to (239.44, 44.66, 125.68) mm, rotated rx -180 ry 0 rz -180 deg; joints [-155.84, -68.496, -48.335, 44.822, 35.494, -38.977]
  Call Extruder(603.09774)
  MoveL 8944 to (239.5, 44.85, 125.68) mm, rotated rx 180 ry 0 rz 180 deg; joints [-155.826, -68.515, -48.297, 44.861, 35.489, -39.017]
  MoveL 8945 to (239.5, 44.85, 125.68) mm, rotated rx 180 ry 0 rz 180 deg; joints [-155.826, -68.515, -48.297, 44.861, 35.489, -39.017]
  Call Extruder(603.21053)
  MoveL 8946 to (239.56, 45.03, 125.68) mm, rotated rx 180 ry 0 rz 180 deg; joints [-155.811, -68.533, -48.259, 44.899, 35.484, -39.056]
  MoveL 8947 to (239.56, 45.03, 125.68) mm, rotated rx 180 ry 0 rz 180 deg; joints [-155.811, -68.533, -48.259, 44.899, 35.484, -39.056]
  Call Extruder(603.32287)
  MoveL 8948 to (239.62, 45.22, 125.68) mm, rotated rx 180 ry 0 rz -180 deg; joints [-155.797, -68.552, -48.221, 44.938, 35.48, -39.096]
  MoveL 8949 to (239.62, 45.22, 125.68) mm, rotated rx 180 ry 0 rz -180 deg; joints [-155.797, -68.552, -48.221, 44.938, 35.48, -39.096]
  Call Extruder(603.43477)
  MoveL 8950 to (239.68, 45.41, 125.68) mm, rotated rx 180 ry 0 rz 180 deg; joints [-155.783, -68.57, -48.183, 44.977, 35.475, -39.135]
  MoveL 8951 to (239.68, 45.41, 125.68) mm, rotated rx 180 ry 0 rz 180 deg; joints [-155.783, -68.57, -48.183, 44.977, 35.475, -39.135]
  Call Extruder(603.55618)
  MoveL 8952 to (239.75, 45.62, 125.68) mm, rotated rx 180 ry 0 rz 180 deg; joints [-155.767, -68.59, -48.142, 45.019, 35.47, -39.178]
  MoveL 8953 to (239.75, 45.62, 125.68) mm, rotated rx 180 ry 0 rz 180 deg; joints [-155.767, -68.59, -48.142, 45.019, 35.47, -39.178]
  Call Extruder(603.68697)
  MoveL 8954 to (239.81, 45.84, 125.68) mm, rotated rx -180 ry 0 rz 180 deg; joints [-155.75, -68.612, -48.097, 45.064, 35.465, -39.225]
  MoveL 8955 to (239.81, 45.84, 125.68) mm, rotated rx -180 ry 0 rz 180 deg; joints [-155.75, -68.612, -48.097, 45.064, 35.465, -39.225]
  Call Extruder(603.81719)
  MoveL 8956 to (239.88, 46.06, 125.68) mm, rotated rx 180 ry 0 rz 180 deg; joints [-155.733, -68.633, -48.054, 45.11, 35.46, -39.271]
  MoveL 8957 to (239.88, 46.06, 125.68) mm, rotated rx 180 ry 0 rz 180 deg; joints [-155.733, -68.633, -48.054, 45.11, 35.46, -39.271]
  Call Extruder(603.94685)
  MoveL 8958 to (239.95, 46.29, 125.68) mm, rotated rx 180 ry 0 rz 180 deg; joints [-155.715, -68.655, -48.009, 45.155, 35.454, -39.318]
  MoveL 8959 to (239.95, 46.29, 125.68) mm, rotated rx 180 ry 0 rz 180 deg; joints [-155.715, -68.655, -48.009, 45.155, 35.454, -39.318]
  Call Extruder(604.07595)
  MoveL 8960 to (240.02, 46.51, 125.68) mm, rotated rx 180 ry 0 rz 180 deg; joints [-155.698, -68.676, -47.965, 45.201, 35.449, -39.364]
  MoveL 8961 to (240.02, 46.51, 125.68) mm, rotated rx 180 ry 0 rz 180 deg; joints [-155.698, -68.676, -47.965, 45.201, 35.449, -39.364]
  Call Extruder(604.19100)
  MoveL 8962 to (240.06, 46.72, 125.68) mm, rotated rx 180 ry 0 rz -180 deg; joints [-155.682, -68.694, -47.929, 45.241, 35.447, -39.404]
  MoveL 8963 to (240.06, 46.72, 125.68) mm, rotated rx 180 ry 0 rz -180 deg; joints [-155.682, -68.694, -47.929, 45.241, 35.447, -39.404]
  Call Extruder(604.30560)
  MoveL 8964 to (240.11, 46.92, 125.68) mm, rotated rx 180 ry 0 rz -180 deg; joints [-155.665, -68.711, -47.893, 45.281, 35.444, -39.445]
  MoveL 8965 to (240.11, 46.92, 125.68) mm, rotated rx 180 ry 0 rz -180 deg; joints [-155.665, -68.711, -47.893, 45.281, 35.444, -39.445]
  Call Extruder(604.41975)
  MoveL 8966 to (240.15, 47.12, 125.68) mm, rotated rx 180 ry 0 rz 180 deg; joints [-155.649, -68.729, -47.857, 45.321, 35.442, -39.485]
  MoveL 8967 to (240.15, 47.12, 125.68) mm, rotated rx 180 ry 0 rz 180 deg; joints [-155.649, -68.729, -47.857, 45.321, 35.442, -39.485]
  Call Extruder(604.53345)
  MoveL 8968 to (240.2, 47.33, 125.68) mm, rotated rx 180 ry 0 rz 180 deg; joints [-155.633, -68.746, -47.821, 45.362, 35.439, -39.526]
  MoveL 8969 to (240.2, 47.33, 125.68) mm, rotated rx 180 ry 0 rz 180 deg; joints [-155.633, -68.746, -47.821, 45.362, 35.439, -39.526]
  Call Extruder(604.65886)
  MoveL 8970 to (240.24, 47.55, 125.68) mm, rotated rx 180 ry 0 rz 180 deg; joints [-155.614, -68.765, -47.782, 45.406, 35.436, -39.57]
  MoveL 8971 to (240.24, 47.55, 125.68) mm, rotated rx 180 ry 0 rz 180 deg; joints [-155.614, -68.765, -47.782, 45.406, 35.436, -39.57]
  Call Extruder(604.79583)
  MoveL 8972 to (240.29, 47.8, 125.68) mm, rotated rx 180 ry 0 rz 180 deg; joints [-155.594, -68.786, -47.739, 45.455, 35.434, -39.619]
  MoveL 8973 to (240.29, 47.8, 125.68) mm, rotated rx 180 ry 0 rz 180 deg; joints [-155.594, -68.786, -47.739, 45.455, 35.434, -39.619]
  Call Extruder(604.93220)
  MoveL 8974 to (240.34, 48.05, 125.68) mm, rotated rx -180 ry 0 rz 180 deg; joints [-155.574, -68.807, -47.697, 45.504, 35.431, -39.668]
  MoveL 8975 to (240.34, 48.05, 125.68) mm, rotated rx -180 ry 0 rz 180 deg; joints [-155.574, -68.807, -47.697, 45.504, 35.431, -39.668]
  Call Extruder(605.06796)
  MoveL 8976 to (240.39, 48.3, 125.68) mm, rotated rx 180 ry 0 rz 180 deg; joints [-155.554, -68.828, -47.654, 45.552, 35.429, -39.717]
  MoveL 8977 to (240.39, 48.3, 125.68) mm, rotated rx 180 ry 0 rz 180 deg; joints [-155.554, -68.828, -47.654, 45.552, 35.429, -39.717]
  Call Extruder(605.20311)
  MoveL 8978 to (240.44, 48.55, 125.68) mm, rotated rx 180 ry 0 rz 180 deg; joints [-155.534, -68.849, -47.611, 45.601, 35.426, -39.765]
  MoveL 8979 to (240.44, 48.55, 125.68) mm, rotated rx 180 ry 0 rz 180 deg; joints [-155.534, -68.849, -47.611, 45.601, 35.426, -39.765]
  Call Extruder(605.33764)
  MoveL 8980 to (240.49, 48.8, 125.68) mm, rotated rx -180 ry 0 rz -180 deg; joints [-155.514, -68.869, -47.568, 45.65, 35.424, -39.814]
  MoveL 8981 to (240.49, 48.8, 125.68) mm, rotated rx -180 ry 0 rz -180 deg; joints [-155.514, -68.869, -47.568, 45.65, 35.424, -39.814]
  Call Extruder(605.47157)
  MoveL 8982 to (240.54, 49.05, 125.68) mm, rotated rx 180 ry 0 rz 180 deg; joints [-155.494, -68.89, -47.525, 45.699, 35.421, -39.863]
  MoveL 8983 to (240.54, 49.05, 125.68) mm, rotated rx 180 ry 0 rz 180 deg; joints [-155.494, -68.89, -47.525, 45.699, 35.421, -39.863]
  Call Extruder(605.61944)
  MoveL 8984 to (240.59, 49.33, 125.68) mm, rotated rx 180 ry 0 rz 180 deg; joints [-155.471, -68.913, -47.479, 45.752, 35.419, -39.917]
  MoveL 8985 to (240.59, 49.33, 125.68) mm, rotated rx 180 ry 0 rz 180 deg; joints [-155.471, -68.913, -47.479, 45.752, 35.419, -39.917]
  Call Extruder(605.78118)
  MoveL 8986 to (240.64, 49.63, 125.68) mm, rotated rx 180 ry 0 rz -180 deg; joints [-155.446, -68.937, -47.429, 45.811, 35.417, -39.975]
  MoveL 8987 to (240.64, 49.63, 125.68) mm, rotated rx 180 ry 0 rz -180 deg; joints [-155.446, -68.937, -47.429, 45.811, 35.417, -39.975]
  Call Extruder(605.94220)
  MoveL 8988 to (240.69, 49.94, 125.68) mm, rotated rx -180 ry 0 rz -180 deg; joints [-155.421, -68.961, -47.38, 45.87, 35.416, -40.034]
  MoveL 8989 to (240.69, 49.94, 125.68) mm, rotated rx -180 ry 0 rz -180 deg; joints [-155.421, -68.961, -47.38, 45.87, 35.416, -40.034]
  Call Extruder(606.10249)
  MoveL 8990 to (240.74, 50.24, 125.68) mm, rotated rx -180 ry 0 rz 180 deg; joints [-155.396, -68.985, -47.33, 45.929, 35.414, -40.093]
  MoveL 8991 to (240.74, 50.24, 125.68) mm, rotated rx -180 ry 0 rz 180 deg; joints [-155.396, -68.985, -47.33, 45.929, 35.414, -40.093]
  Call Extruder(606.26205)
  MoveL 8992 to (240.78, 50.55, 125.68) mm, rotated rx 180 ry 0 rz 180 deg; joints [-155.371, -69.01, -47.28, 45.988, 35.413, -40.151]
  MoveL 8993 to (240.78, 50.55, 125.68) mm, rotated rx 180 ry 0 rz 180 deg; joints [-155.371, -69.01, -47.28, 45.988, 35.413, -40.151]
  Call Extruder(606.42088)
  MoveL 8994 to (240.83, 50.86, 125.68) mm, rotated rx -180 ry 0 rz -180 deg; joints [-155.346, -69.034, -47.23, 46.047, 35.411, -40.21]
  MoveL 8995 to (240.83, 50.86, 125.68) mm, rotated rx -180 ry 0 rz -180 deg; joints [-155.346, -69.034, -47.23, 46.047, 35.411, -40.21]
  Call Extruder(606.59956)
  MoveL 8996 to (240.88, 51.2, 125.68) mm, rotated rx 180 ry 0 rz 180 deg; joints [-155.317, -69.06, -47.176, 46.113, 35.41, -40.276]
  MoveL 8997 to (240.88, 51.2, 125.68) mm, rotated rx 180 ry 0 rz 180 deg; joints [-155.317, -69.06, -47.176, 46.113, 35.41, -40.276]
  Call Extruder(606.79800)
  MoveL 8998 to (240.92, 51.59, 125.68) mm, rotated rx 180 ry 0 rz -180 deg; joints [-155.285, -69.089, -47.116, 46.187, 35.41, -40.348]
  MoveL 8999 to (240.92, 51.59, 125.68) mm, rotated rx 180 ry 0 rz -180 deg; joints [-155.285, -69.089, -47.116, 46.187, 35.41, -40.348]
  Call Extruder(606.99557)
  MoveL 9000 to (240.97, 51.98, 125.68) mm, rotated rx -180 ry 0 rz 180 deg; joints [-155.252, -69.118, -47.057, 46.26, 35.41, -40.421]
  MoveL 9001 to (240.97, 51.98, 125.68) mm, rotated rx -180 ry 0 rz 180 deg; joints [-155.252, -69.118, -47.057, 46.26, 35.41, -40.421]
  Call Extruder(607.19228)
  MoveL 9002 to (241.02, 52.36, 125.68) mm, rotated rx 180 ry 0 rz 180 deg; joints [-155.22, -69.147, -46.997, 46.334, 35.41, -40.494]
  MoveL 9003 to (241.02, 52.36, 125.68) mm, rotated rx 180 ry 0 rz 180 deg; joints [-155.22, -69.147, -46.997, 46.334, 35.41, -40.494]
  Call Extruder(607.38812)
  MoveL 9004 to (241.06, 52.75, 125.68) mm, rotated rx 180 ry 0 rz 180 deg; joints [-155.188, -69.176, -46.938, 46.407, 35.41, -40.566]
  MoveL 9005 to (241.06, 52.75, 125.68) mm, rotated rx 180 ry 0 rz 180 deg; joints [-155.188, -69.176, -46.938, 46.407, 35.41, -40.566]
  Call Extruder(607.68356)
  MoveL 9006 to (241.11, 53.34, 125.68) mm, rotated rx 180 ry 0 rz 180 deg; joints [-155.138, -69.218, -46.853, 46.517, 35.412, -40.674]
  MoveL 9007 to (241.11, 53.34, 125.68) mm, rotated rx 180 ry 0 rz 180 deg; joints [-155.138, -69.218, -46.853, 46.517, 35.412, -40.674]
  Call Extruder(607.97766)
  MoveL 9008 to (241.16, 53.93, 125.68) mm, rotated rx 180 ry 0 rz 180 deg; joints [-155.088, -69.259, -46.768, 46.627, 35.415, -40.782]
  MoveL 9009 to (241.16, 53.93, 125.68) mm, rotated rx 180 ry 0 rz 180 deg; joints [-155.088, -69.259, -46.768, 46.627, 35.415, -40.782]
  Call Extruder(608.27044)
  MoveL 9010 to (241.2, 54.52, 125.68) mm, rotated rx -180 ry 0 rz 180 deg; joints [-155.038, -69.301, -46.683, 46.737, 35.417, -40.89]
  MoveL 9011 to (241.2, 54.52, 125.68) mm, rotated rx -180 ry 0 rz 180 deg; joints [-155.038, -69.301, -46.683, 46.737, 35.417, -40.89]
  Call Extruder(608.84389)
  MoveL 9012 to (241.25, 55.68, 125.68) mm, rotated rx 180 ry 0 rz 180 deg; joints [-154.938, -69.377, -46.526, 46.949, 35.428, -41.097]
  MoveL 9013 to (241.25, 55.68, 125.68) mm, rotated rx 180 ry 0 rz 180 deg; joints [-154.938, -69.377, -46.526, 46.949, 35.428, -41.097]
  Call Extruder(609.55772)
  MoveL 9014 to (241.29, 57.14, 125.68) mm, rotated rx 180 ry 0 rz 180 deg; joints [-154.812, -69.471, -46.334, 47.214, 35.444, -41.355]
  Call Extruder(651.62260)
  MoveL 9015 to (241.29, 142.86, 125.68) mm, rotated rx -180 ry 0 rz 180 deg; joints [-147.778, -76.212, -32.684, 62.804, 36.832, -57.301]
  Call Extruder(652.05103)
  MoveL 9016 to (241.27, 143.73, 125.68) mm, rotated rx 180 ry 0 rz 180 deg; joints [-147.711, -76.298, -32.513, 62.967, 36.85, -57.476]
  MoveL 9017 to (241.27, 143.73, 125.68) mm, rotated rx 180 ry 0 rz 180 deg; joints [-147.711, -76.298, -32.513, 62.967, 36.85, -57.476]
  Call Extruder(652.62448)
  MoveL 9018 to (241.22, 144.9, 125.68) mm, rotated rx 180 ry 0 rz 180 deg; joints [-147.62, -76.409, -32.291, 63.18, 36.876, -57.706]
  MoveL 9019 to (241.22, 144.9, 125.68) mm, rotated rx 180 ry 0 rz 180 deg; joints [-147.62, -76.409, -32.291, 63.18, 36.876, -57.706]
  Call Extruder(653.05882)
  MoveL 9020 to (241.18, 145.77, 125.68) mm, rotated rx 180 ry 0 rz 180 deg; joints [-147.551, -76.491, -32.127, 63.339, 36.898, -57.877]
  MoveL 9021 to (241.18, 145.77, 125.68) mm, rotated rx 180 ry 0 rz 180 deg; joints [-147.551, -76.491, -32.127, 63.339, 36.898, -57.877]
  Call Extruder(653.35293)
  MoveL 9022 to (241.13, 146.36, 125.68) mm, rotated rx 180 ry 0 rz -180 deg; joints [-147.504, -76.544, -32.021, 63.443, 36.914, -57.989]
  MoveL 9023 to (241.13, 146.36, 125.68) mm, rotated rx 180 ry 0 rz -180 deg; joints [-147.504, -76.544, -32.021, 63.443, 36.914, -57.989]
  Call Extruder(653.64837)
  MoveL 9024 to (241.09, 146.95, 125.68) mm, rotated rx -180 ry 0 rz -180 deg; joints [-147.457, -76.597, -31.914, 63.548, 36.93, -58.102]
  MoveL 9025 to (241.09, 146.95, 125.68) mm, rotated rx -180 ry 0 rz -180 deg; joints [-147.457, -76.597, -31.914, 63.548, 36.93, -58.102]
  Call Extruder(653.89462)
  MoveL 9026 to (241.04, 147.44, 125.68) mm, rotated rx 180 ry 0 rz 180 deg; joints [-147.417, -76.64, -31.828, 63.634, 36.944, -58.194]
  MoveL 9027 to (241.04, 147.44, 125.68) mm, rotated rx 180 ry 0 rz 180 deg; joints [-147.417, -76.64, -31.828, 63.634, 36.944, -58.194]
  Call Extruder(654.09133)
  MoveL 9028 to (240.99, 147.83, 125.68) mm, rotated rx 180 ry 0 rz 180 deg; joints [-147.386, -76.673, -31.763, 63.701, 36.957, -58.265]
  MoveL 9029 to (240.99, 147.83, 125.68) mm, rotated rx 180 ry 0 rz 180 deg; joints [-147.386, -76.673, -31.763, 63.701, 36.957, -58.265]
  Call Extruder(654.28890)
  MoveL 9030 to (240.95, 148.22, 125.68) mm, rotated rx 180 ry 0 rz 180 deg; joints [-147.354, -76.706, -31.697, 63.768, 36.969, -58.335]
  MoveL 9031 to (240.95, 148.22, 125.68) mm, rotated rx 180 ry 0 rz 180 deg; joints [-147.354, -76.706, -31.697, 63.768, 36.969, -58.335]
  Call Extruder(654.48734)
  MoveL 9032 to (240.9, 148.6, 125.68) mm, rotated rx 180 ry 0 rz -180 deg; joints [-147.322, -76.739, -31.631, 63.834, 36.982, -58.407]
  MoveL 9033 to (240.9, 148.6, 125.68) mm, rotated rx 180 ry 0 rz -180 deg; joints [-147.322, -76.739, -31.631, 63.834, 36.982, -58.407]
  Call Extruder(654.68665)
  MoveL 9034 to (240.86, 148.99, 125.68) mm, rotated rx -180 ry 0 rz 180 deg; joints [-147.291, -76.772, -31.565, 63.901, 36.994, -58.478]
  MoveL 9035 to (240.86, 148.99, 125.68) mm, rotated rx -180 ry 0 rz 180 deg; joints [-147.291, -76.772, -31.565, 63.901, 36.994, -58.478]
  Call Extruder(654.84549)
  MoveL 9036 to (240.81, 149.3, 125.68) mm, rotated rx -180 ry 0 rz 180 deg; joints [-147.265, -76.796, -31.517, 63.952, 37.005, -58.531]
  MoveL 9037 to (240.81, 149.3, 125.68) mm, rotated rx -180 ry 0 rz 180 deg; joints [-147.265, -76.796, -31.517, 63.952, 37.005, -58.531]
  Call Extruder(655.00505)
  MoveL 9038 to (240.76, 149.6, 125.68) mm, rotated rx 180 ry 0 rz 180 deg; joints [-147.24, -76.82, -31.469, 64.003, 37.016, -58.585]
  MoveL 9039 to (240.76, 149.6, 125.68) mm, rotated rx 180 ry 0 rz 180 deg; joints [-147.24, -76.82, -31.469, 64.003, 37.016, -58.585]
  Call Extruder(655.16534)
  MoveL 9040 to (240.71, 149.91, 125.68) mm, rotated rx -180 ry 0 rz -180 deg; joints [-147.214, -76.844, -31.42, 64.054, 37.028, -58.639]
  MoveL 9041 to (240.71, 149.91, 125.68) mm, rotated rx -180 ry 0 rz -180 deg; joints [-147.214, -76.844, -31.42, 64.054, 37.028, -58.639]
  Call Extruder(655.32635)
  MoveL 9042 to (240.66, 150.21, 125.68) mm, rotated rx -180 ry 0 rz -180 deg; joints [-147.189, -76.868, -31.372, 64.104, 37.039, -58.692]
  MoveL 9043 to (240.66, 150.21, 125.68) mm, rotated rx -180 ry 0 rz -180 deg; joints [-147.189, -76.868, -31.372, 64.104, 37.039, -58.692]
  Call Extruder(655.48810)
  MoveL 9044 to (240.61, 150.52, 125.68) mm, rotated rx -180 ry 0 rz 180 deg; joints [-147.163, -76.893, -31.323, 64.155, 37.05, -58.746]
  MoveL 9045 to (240.61, 150.52, 125.68) mm, rotated rx -180 ry 0 rz 180 deg; joints [-147.163, -76.893, -31.323, 64.155, 37.05, -58.746]
  Call Extruder(655.65057)
  MoveL 9046 to (240.56, 150.83, 125.68) mm, rotated rx -180 ry 0 rz -180 deg; joints [-147.138, -76.917, -31.275, 64.206, 37.061, -58.8]
  MoveL 9047 to (240.56, 150.83, 125.68) mm, rotated rx -180 ry 0 rz -180 deg; joints [-147.138, -76.917, -31.275, 64.206, 37.061, -58.8]
  Call Extruder(655.78449)
  MoveL 9048 to (240.52, 151.07, 125.68) mm, rotated rx 180 ry 0 rz 180 deg; joints [-147.117, -76.936, -31.238, 64.246, 37.071, -58.842]
  MoveL 9049 to (240.52, 151.07, 125.68) mm, rotated rx 180 ry 0 rz 180 deg; joints [-147.117, -76.936, -31.238, 64.246, 37.071, -58.842]
  Call Extruder(655.91903)
  MoveL 9050 to (240.47, 151.32, 125.68) mm, rotated rx 180 ry 0 rz -180 deg; joints [-147.095, -76.954, -31.202, 64.286, 37.082, -58.883]
  MoveL 9051 to (240.47, 151.32, 125.68) mm, rotated rx 180 ry 0 rz -180 deg; joints [-147.095, -76.954, -31.202, 64.286, 37.082, -58.883]
  Call Extruder(656.05418)
  MoveL 9052 to (240.42, 151.57, 125.68) mm, rotated rx -180 ry 0 rz 180 deg; joints [-147.074, -76.972, -31.165, 64.326, 37.092, -58.925]
  MoveL 9053 to (240.42, 151.57, 125.68) mm, rotated rx -180 ry 0 rz 180 deg; joints [-147.074, -76.972, -31.165, 64.326, 37.092, -58.925]
  Call Extruder(656.18994)
  MoveL 9054 to (240.37, 151.82, 125.68) mm, rotated rx -180 ry 0 rz -180 deg; joints [-147.053, -76.99, -31.128, 64.366, 37.102, -58.967]
  MoveL 9055 to (240.37, 151.82, 125.68) mm, rotated rx -180 ry 0 rz -180 deg; joints [-147.053, -76.99, -31.128, 64.366, 37.102, -58.967]
  Call Extruder(656.32630)
  MoveL 9056 to (240.32, 152.07, 125.68) mm, rotated rx -180 ry 0 rz 180 deg; joints [-147.032, -77.009, -31.092, 64.406, 37.112, -59.009]
  MoveL 9057 to (240.32, 152.07, 125.68) mm, rotated rx -180 ry 0 rz 180 deg; joints [-147.032, -77.009, -31.092, 64.406, 37.112, -59.009]
  Call Extruder(656.46328)
  MoveL 9058 to (240.27, 152.32, 125.68) mm, rotated rx -180 ry 0 rz 180 deg; joints [-147.011, -77.027, -31.055, 64.446, 37.123, -59.051]
  MoveL 9059 to (240.27, 152.32, 125.68) mm, rotated rx -180 ry 0 rz 180 deg; joints [-147.011, -77.027, -31.055, 64.446, 37.123, -59.051]
  Call Extruder(656.60087)
  MoveL 9060 to (240.22, 152.57, 125.68) mm, rotated rx 180 ry 0 rz 180 deg; joints [-146.989, -77.046, -31.018, 64.486, 37.133, -59.092]
  MoveL 9061 to (240.22, 152.57, 125.68) mm, rotated rx 180 ry 0 rz 180 deg; joints [-146.989, -77.046, -31.018, 64.486, 37.133, -59.092]
  Call Extruder(656.71457)
  MoveL 9062 to (240.17, 152.77, 125.68) mm, rotated rx 180 ry 0 rz 180 deg; joints [-146.972, -77.06, -30.989, 64.518, 37.142, -59.126]
  MoveL 9063 to (240.17, 152.77, 125.68) mm, rotated rx 180 ry 0 rz 180 deg; joints [-146.972, -77.06, -30.989, 64.518, 37.142, -59.126]
  Call Extruder(656.82872)
  MoveL 9064 to (240.13, 152.98, 125.68) mm, rotated rx -180 ry 0 rz -180 deg; joints [-146.954, -77.075, -30.96, 64.55, 37.151, -59.159]
  MoveL 9065 to (240.13, 152.98, 125.68) mm, rotated rx -180 ry 0 rz -180 deg; joints [-146.954, -77.075, -30.96, 64.55, 37.151, -59.159]
  Call Extruder(656.94332)
  MoveL 9066 to (240.08, 153.18, 125.68) mm, rotated rx 180 ry 0 rz 180 deg; joints [-146.937, -77.089, -30.931, 64.582, 37.16, -59.193]
  MoveL 9067 to (240.08, 153.18, 125.68) mm, rotated rx 180 ry 0 rz 180 deg; joints [-146.937, -77.089, -30.931, 64.582, 37.16, -59.193]
  Call Extruder(657.05837)
  MoveL 9068 to (240.04, 153.39, 125.68) mm, rotated rx 180 ry 0 rz -180 deg; joints [-146.919, -77.104, -30.902, 64.614, 37.168, -59.226]
  MoveL 9069 to (240.04, 153.39, 125.68) mm, rotated rx 180 ry 0 rz -180 deg; joints [-146.919, -77.104, -30.902, 64.614, 37.168, -59.226]
  Call Extruder(657.18060)
  MoveL 9070 to (239.98, 153.6, 125.68) mm, rotated rx 180 ry 0 rz -180 deg; joints [-146.9, -77.117, -30.875, 64.647, 37.179, -59.26]
  MoveL 9071 to (239.98, 153.6, 125.68) mm, rotated rx 180 ry 0 rz -180 deg; joints [-146.9, -77.117, -30.875, 64.647, 37.179, -59.26]
  Call Extruder(657.31026)
  MoveL 9072 to (239.92, 153.82, 125.68) mm, rotated rx 180 ry 0 rz 180 deg; joints [-146.88, -77.13, -30.849, 64.679, 37.191, -59.292]
  MoveL 9073 to (239.92, 153.82, 125.68) mm, rotated rx 180 ry 0 rz 180 deg; joints [-146.88, -77.13, -30.849, 64.679, 37.191, -59.292]
  Call Extruder(657.44048)
  MoveL 9074 to (239.85, 154.05, 125.68) mm, rotated rx -180 ry 0 rz 180 deg; joints [-146.86, -77.143, -30.824, 64.711, 37.202, -59.325]
  MoveL 9075 to (239.85, 154.05, 125.68) mm, rotated rx -180 ry 0 rz 180 deg; joints [-146.86, -77.143, -30.824, 64.711, 37.202, -59.325]
  Call Extruder(657.57127)
  MoveL 9076 to (239.78, 154.27, 125.68) mm, rotated rx -180 ry 0 rz -180 deg; joints [-146.84, -77.156, -30.797, 64.744, 37.214, -59.358]
  MoveL 9077 to (239.78, 154.27, 125.68) mm, rotated rx -180 ry 0 rz -180 deg; joints [-146.84, -77.156, -30.797, 64.744, 37.214, -59.358]
  Call Extruder(657.70262)
  MoveL 9078 to (239.71, 154.49, 125.68) mm, rotated rx 180 ry 0 rz 180 deg; joints [-146.82, -77.169, -30.772, 64.776, 37.226, -59.391]
  MoveL 9079 to (239.71, 154.49, 125.68) mm, rotated rx 180 ry 0 rz 180 deg; joints [-146.82, -77.169, -30.772, 64.776, 37.226, -59.391]
  Call Extruder(657.81453)
  MoveL 9080 to (239.65, 154.68, 125.68) mm, rotated rx -180 ry 0 rz -180 deg; joints [-146.803, -77.179, -30.751, 64.802, 37.236, -59.417]
  MoveL 9081 to (239.65, 154.68, 125.68) mm, rotated rx -180 ry 0 rz -180 deg; joints [-146.803, -77.179, -30.751, 64.802, 37.236, -59.417]
  Call Extruder(657.92687)
  MoveL 9082 to (239.59, 154.87, 125.68) mm, rotated rx -180 ry 0 rz 180 deg; joints [-146.785, -77.19, -30.731, 64.829, 37.247, -59.444]
  MoveL 9083 to (239.59, 154.87, 125.68) mm, rotated rx -180 ry 0 rz 180 deg; joints [-146.785, -77.19, -30.731, 64.829, 37.247, -59.444]
  Call Extruder(658.03966)
  MoveL 9084 to (239.53, 155.06, 125.68) mm, rotated rx 180 ry 0 rz -180 deg; joints [-146.768, -77.2, -30.71, 64.855, 37.257, -59.471]
  MoveL 9085 to (239.53, 155.06, 125.68) mm, rotated rx 180 ry 0 rz -180 deg; joints [-146.768, -77.2, -30.71, 64.855, 37.257, -59.471]
  Call Extruder(658.15290)
  MoveL 9086 to (239.47, 155.25, 125.68) mm, rotated rx 180 ry 0 rz 180 deg; joints [-146.751, -77.21, -30.69, 64.882, 37.268, -59.498]
  MoveL 9087 to (239.47, 155.25, 125.68) mm, rotated rx 180 ry 0 rz 180 deg; joints [-146.751, -77.21, -30.69, 64.882, 37.268, -59.498]
  Call Extruder(658.26658)
  MoveL 9088 to (239.41, 155.44, 125.68) mm, rotated rx -180 ry 0 rz -180 deg; joints [-146.734, -77.221, -30.669, 64.909, 37.278, -59.524]
  MoveL 9089 to (239.41, 155.44, 125.68) mm, rotated rx -180 ry 0 rz -180 deg; joints [-146.734, -77.221, -30.669, 64.909, 37.278, -59.524]
  Call Extruder(658.44854)
  MoveL 9090 to (239.29, 155.73, 125.68) mm, rotated rx -180 ry 0 rz 180 deg; joints [-146.706, -77.232, -30.646, 64.946, 37.297, -59.56]
  MoveL 9091 to (239.29, 155.73, 125.68) mm, rotated rx -180 ry 0 rz 180 deg; joints [-146.706, -77.232, -30.646, 64.946, 37.297, -59.56]
  Call Extruder(658.63125)
  MoveL 9092 to (239.17, 156.02, 125.68) mm, rotated rx -180 ry 0 rz 180 deg; joints [-146.678, -77.244, -30.622, 64.983, 37.316, -59.596]
  MoveL 9093 to (239.17, 156.02, 125.68) mm, rotated rx -180 ry 0 rz 180 deg; joints [-146.678, -77.244, -30.622, 64.983, 37.316, -59.596]
  Call Extruder(658.80168)
  MoveL 9094 to (239.05, 156.29, 125.68) mm, rotated rx 180 ry 0 rz 180 deg; joints [-146.652, -77.255, -30.601, 65.017, 37.334, -59.629]
  MoveL 9095 to (239.05, 156.29, 125.68) mm, rotated rx 180 ry 0 rz 180 deg; joints [-146.652, -77.255, -30.601, 65.017, 37.334, -59.629]
  Call Extruder(658.95972)
  MoveL 9096 to (238.94, 156.54, 125.68) mm, rotated rx -180 ry 0 rz -180 deg; joints [-146.628, -77.264, -30.582, 65.048, 37.351, -59.659]
  MoveL 9097 to (238.94, 156.54, 125.68) mm, rotated rx -180 ry 0 rz -180 deg; joints [-146.628, -77.264, -30.582, 65.048, 37.351, -59.659]
  Call Extruder(659.11835)
  MoveL 9098 to (238.84, 156.79, 125.68) mm, rotated rx 180 ry 0 rz 180 deg; joints [-146.604, -77.273, -30.564, 65.079, 37.367, -59.689]
  MoveL 9099 to (238.84, 156.79, 125.68) mm, rotated rx 180 ry 0 rz 180 deg; joints [-146.604, -77.273, -30.564, 65.079, 37.367, -59.689]
  Call Extruder(659.32451)
  MoveL 9100 to (238.66, 157.09, 125.68) mm, rotated rx 180 ry 0 rz 180 deg; joints [-146.573, -77.278, -30.555, 65.11, 37.393, -59.716]
  MoveL 9101 to (238.66, 157.09, 125.68) mm, rotated rx 180 ry 0 rz 180 deg; joints [-146.573, -77.278, -30.555, 65.11, 37.393, -59.716]
  Call Extruder(659.53144)
  MoveL 9102 to (238.49, 157.4, 125.68) mm, rotated rx 180 ry 0 rz -180 deg; joints [-146.542, -77.282, -30.547, 65.141, 37.418, -59.743]
  MoveL 9103 to (238.49, 157.4, 125.68) mm, rotated rx 180 ry 0 rz -180 deg; joints [-146.542, -77.282, -30.547, 65.141, 37.418, -59.743]
  Call Extruder(659.73916)
  MoveL 9104 to (238.31, 157.7, 125.68) mm, rotated rx 180 ry 0 rz -180 deg; joints [-146.51, -77.286, -30.538, 65.172, 37.444, -59.77]
  MoveL 9105 to (238.31, 157.7, 125.68) mm, rotated rx 180 ry 0 rz -180 deg; joints [-146.51, -77.286, -30.538, 65.172, 37.444, -59.77]
  Call Extruder(659.94765)
  MoveL 9106 to (238.14, 158.01, 125.68) mm, rotated rx -180 ry 0 rz 180 deg; joints [-146.479, -77.29, -30.53, 65.203, 37.469, -59.797]
  MoveL 9107 to (238.14, 158.01, 125.68) mm, rotated rx -180 ry 0 rz 180 deg; joints [-146.479, -77.29, -30.53, 65.203, 37.469, -59.797]
  Call Extruder(660.12717)
  MoveL 9108 to (237.96, 158.25, 125.68) mm, rotated rx -180 ry 0 rz 180 deg; joints [-146.452, -77.288, -30.535, 65.223, 37.493, -59.811]
  MoveL 9109 to (237.96, 158.25, 125.68) mm, rotated rx -180 ry 0 rz 180 deg; joints [-146.452, -77.288, -30.535, 65.223, 37.493, -59.811]
  Call Extruder(660.46059)
  MoveL 9110 to (237.63, 158.7, 125.68) mm, rotated rx 180 ry 0 rz 180 deg; joints [-146.402, -77.283, -30.544, 65.259, 37.538, -59.837]
  MoveL 9111 to (237.63, 158.7, 125.68) mm, rotated rx 180 ry 0 rz 180 deg; joints [-146.402, -77.283, -30.544, 65.259, 37.538, -59.837]
  Call Extruder(660.79519)
  MoveL 9112 to (237.3, 159.15, 125.68) mm, rotated rx 180 ry 0 rz 180 deg; joints [-146.352, -77.279, -30.553, 65.295, 37.584, -59.863]
  Call Extruder(661.62314)
  MoveL 9113 to (236.39, 160.19, 125.68) mm, rotated rx -180 ry 0 rz 180 deg; joints [-146.229, -77.242, -30.625, 65.353, 37.705, -59.889]
  Call Extruder(662.45109)
  MoveL 9114 to (235.35, 161.1, 125.68) mm, rotated rx -180 ry 0 rz 180 deg; joints [-146.109, -77.173, -30.765, 65.369, 37.837, -59.863]
  Call Extruder(662.61839)
  MoveL 9115 to (235.13, 161.27, 125.68) mm, rotated rx -180 ry 0 rz 180 deg; joints [-146.086, -77.154, -30.803, 65.367, 37.866, -59.851]
  MoveL 9116 to (235.13, 161.27, 125.68) mm, rotated rx -180 ry 0 rz 180 deg; joints [-146.086, -77.154, -30.803, 65.367, 37.866, -59.851]
  Call Extruder(662.95182)
  MoveL 9117 to (234.68, 161.59, 125.68) mm, rotated rx 180 ry 0 rz 180 deg; joints [-146.039, -77.116, -30.878, 65.361, 37.922, -59.826]
  MoveL 9118 to (234.68, 161.59, 125.68) mm, rotated rx 180 ry 0 rz 180 deg; joints [-146.039, -77.116, -30.878, 65.361, 37.922, -59.826]
  Call Extruder(663.28405)
  MoveL 9119 to (234.22, 161.92, 125.68) mm, rotated rx 180 ry 0 rz 180 deg; joints [-145.992, -77.078, -30.953, 65.356, 37.978, -59.801]
  MoveL 9120 to (234.22, 161.92, 125.68) mm, rotated rx 180 ry 0 rz 180 deg; joints [-145.992, -77.078, -30.953, 65.356, 37.978, -59.801]
  Call Extruder(663.40172)
  MoveL 9121 to (234.05, 162.02, 125.68) mm, rotated rx 180 ry 0 rz 180 deg; joints [-145.976, -77.062, -30.986, 65.35, 37.999, -59.786]
  MoveL 9122 to (234.05, 162.02, 125.68) mm, rotated rx 180 ry 0 rz 180 deg; joints [-145.976, -77.062, -30.986, 65.35, 37.999, -59.786]
  Call Extruder(663.60945)
  MoveL 9123 to (233.75, 162.2, 125.68) mm, rotated rx 180 ry 0 rz 180 deg; joints [-145.947, -77.031, -31.047, 65.338, 38.036, -59.76]
  MoveL 9124 to (233.75, 162.2, 125.68) mm, rotated rx 180 ry 0 rz 180 deg; joints [-145.947, -77.031, -31.047, 65.338, 38.036, -59.76]
  Call Extruder(663.81640)
  MoveL 9125 to (233.45, 162.37, 125.68) mm, rotated rx 180 ry 0 rz -180 deg; joints [-145.919, -77.001, -31.107, 65.326, 38.073, -59.734]
  MoveL 9126 to (233.45, 162.37, 125.68) mm, rotated rx 180 ry 0 rz -180 deg; joints [-145.919, -77.001, -31.107, 65.326, 38.073, -59.734]
  Call Extruder(664.02257)
  MoveL 9127 to (233.14, 162.55, 125.68) mm, rotated rx -180 ry 0 rz 180 deg; joints [-145.891, -76.971, -31.167, 65.315, 38.11, -59.708]
  MoveL 9128 to (233.14, 162.55, 125.68) mm, rotated rx -180 ry 0 rz 180 deg; joints [-145.891, -76.971, -31.167, 65.315, 38.11, -59.708]
  Call Extruder(664.20424)
  MoveL 9129 to (232.86, 162.69, 125.68) mm, rotated rx -180 ry 0 rz 180 deg; joints [-145.866, -76.942, -31.225, 65.301, 38.143, -59.681]
  MoveL 9130 to (232.86, 162.69, 125.68) mm, rotated rx -180 ry 0 rz 180 deg; joints [-145.866, -76.942, -31.225, 65.301, 38.143, -59.681]
  Call Extruder(664.36221)
  MoveL 9131 to (232.62, 162.8, 125.68) mm, rotated rx 180 ry 0 rz -180 deg; joints [-145.845, -76.914, -31.282, 65.285, 38.173, -59.653]
  MoveL 9132 to (232.62, 162.8, 125.68) mm, rotated rx 180 ry 0 rz -180 deg; joints [-145.845, -76.914, -31.282, 65.285, 38.173, -59.653]
  Call Extruder(664.51957)
  MoveL 9133 to (232.37, 162.9, 125.68) mm, rotated rx -180 ry 0 rz 180 deg; joints [-145.825, -76.885, -31.339, 65.269, 38.203, -59.624]
  MoveL 9134 to (232.37, 162.9, 125.68) mm, rotated rx -180 ry 0 rz 180 deg; joints [-145.825, -76.885, -31.339, 65.269, 38.203, -59.624]
  Call Extruder(664.70231)
  MoveL 9135 to (232.07, 163.02, 125.68) mm, rotated rx 180 ry 0 rz 180 deg; joints [-145.801, -76.851, -31.406, 65.25, 38.237, -59.59]
  MoveL 9136 to (232.07, 163.02, 125.68) mm, rotated rx 180 ry 0 rz 180 deg; joints [-145.801, -76.851, -31.406, 65.25, 38.237, -59.59]
  Call Extruder(664.88429)
  MoveL 9137 to (231.78, 163.15, 125.68) mm, rotated rx -180 ry 0 rz -180 deg; joints [-145.777, -76.818, -31.474, 65.23, 38.272, -59.556]
  MoveL 9138 to (231.78, 163.15, 125.68) mm, rotated rx -180 ry 0 rz -180 deg; joints [-145.777, -76.818, -31.474, 65.23, 38.272, -59.556]
  Call Extruder(665.03163)
  MoveL 9139 to (231.54, 163.24, 125.68) mm, rotated rx 180 ry 0 rz 180 deg; joints [-145.759, -76.789, -31.531, 65.213, 38.3, -59.526]
  MoveL 9140 to (231.54, 163.24, 125.68) mm, rotated rx 180 ry 0 rz 180 deg; joints [-145.759, -76.789, -31.531, 65.213, 38.3, -59.526]
  Call Extruder(665.14485)
  MoveL 9141 to (231.35, 163.3, 125.68) mm, rotated rx -180 ry 0 rz 180 deg; joints [-145.744, -76.766, -31.578, 65.198, 38.322, -59.501]
  MoveL 9142 to (231.35, 163.3, 125.68) mm, rotated rx -180 ry 0 rz 180 deg; joints [-145.744, -76.766, -31.578, 65.198, 38.322, -59.501]
  Call Extruder(665.25763)
  MoveL 9143 to (231.17, 163.36, 125.68) mm, rotated rx 180 ry 0 rz 180 deg; joints [-145.73, -76.742, -31.624, 65.183, 38.344, -59.476]
  MoveL 9144 to (231.17, 163.36, 125.68) mm, rotated rx 180 ry 0 rz 180 deg; joints [-145.73, -76.742, -31.624, 65.183, 38.344, -59.476]
  Call Extruder(665.36996)
  MoveL 9145 to (230.98, 163.42, 125.68) mm, rotated rx -180 ry 0 rz 180 deg; joints [-145.716, -76.719, -31.671, 65.167, 38.366, -59.451]
  MoveL 9146 to (230.98, 163.42, 125.68) mm, rotated rx -180 ry 0 rz 180 deg; joints [-145.716, -76.719, -31.671, 65.167, 38.366, -59.451]
  Call Extruder(665.48185)
  MoveL 9147 to (230.79, 163.48, 125.68) mm, rotated rx -180 ry 0 rz 180 deg; joints [-145.702, -76.695, -31.718, 65.152, 38.388, -59.425]
  MoveL 9148 to (230.79, 163.48, 125.68) mm, rotated rx -180 ry 0 rz 180 deg; joints [-145.702, -76.695, -31.718, 65.152, 38.388, -59.425]
  Call Extruder(665.60326)
  MoveL 9149 to (230.58, 163.55, 125.68) mm, rotated rx -180 ry 0 rz 180 deg; joints [-145.687, -76.669, -31.769, 65.135, 38.412, -59.398]
  MoveL 9150 to (230.58, 163.55, 125.68) mm, rotated rx -180 ry 0 rz 180 deg; joints [-145.687, -76.669, -31.769, 65.135, 38.412, -59.398]
  Call Extruder(665.73407)
  MoveL 9151 to (230.36, 163.61, 125.68) mm, rotated rx -180 ry 0 rz 180 deg; joints [-145.67, -76.641, -31.826, 65.116, 38.438, -59.367]
  MoveL 9152 to (230.36, 163.61, 125.68) mm, rotated rx -180 ry 0 rz 180 deg; joints [-145.67, -76.641, -31.826, 65.116, 38.438, -59.367]
  Call Extruder(665.86432)
  MoveL 9153 to (230.14, 163.68, 125.68) mm, rotated rx -180 ry 0 rz 180 deg; joints [-145.654, -76.613, -31.882, 65.098, 38.464, -59.337]
  MoveL 9154 to (230.14, 163.68, 125.68) mm, rotated rx -180 ry 0 rz 180 deg; joints [-145.654, -76.613, -31.882, 65.098, 38.464, -59.337]
  Call Extruder(665.99400)
  MoveL 9155 to (229.91, 163.75, 125.68) mm, rotated rx -180 ry 0 rz 180 deg; joints [-145.638, -76.585, -31.938, 65.079, 38.49, -59.306]
  MoveL 9156 to (229.91, 163.75, 125.68) mm, rotated rx -180 ry 0 rz 180 deg; joints [-145.638, -76.585, -31.938, 65.079, 38.49, -59.306]
  Call Extruder(666.12312)
  MoveL 9157 to (229.69, 163.82, 125.68) mm, rotated rx -180 ry 0 rz -180 deg; joints [-145.621, -76.557, -31.995, 65.06, 38.516, -59.276]
  MoveL 9158 to (229.69, 163.82, 125.68) mm, rotated rx -180 ry 0 rz -180 deg; joints [-145.621, -76.557, -31.995, 65.06, 38.516, -59.276]
  Call Extruder(666.23819)
  MoveL 9159 to (229.48, 163.86, 125.68) mm, rotated rx -180 ry 0 rz -180 deg; joints [-145.607, -76.529, -32.05, 65.04, 38.539, -59.245]
  MoveL 9160 to (229.48, 163.86, 125.68) mm, rotated rx -180 ry 0 rz -180 deg; joints [-145.607, -76.529, -32.05, 65.04, 38.539, -59.245]
  Call Extruder(666.35282)
  MoveL 9161 to (229.28, 163.91, 125.68) mm, rotated rx -180 ry 0 rz -180 deg; joints [-145.594, -76.502, -32.104, 65.021, 38.562, -59.214]
  MoveL 9162 to (229.28, 163.91, 125.68) mm, rotated rx -180 ry 0 rz -180 deg; joints [-145.594, -76.502, -32.104, 65.021, 38.562, -59.214]
  Call Extruder(666.46699)
  MoveL 9163 to (229.08, 163.95, 125.68) mm, rotated rx -180 ry 0 rz 180 deg; joints [-145.58, -76.475, -32.159, 65.001, 38.586, -59.183]
  MoveL 9164 to (229.08, 163.95, 125.68) mm, rotated rx -180 ry 0 rz 180 deg; joints [-145.58, -76.475, -32.159, 65.001, 38.586, -59.183]
  Call Extruder(666.58070)
  MoveL 9165 to (228.87, 164, 125.68) mm, rotated rx 180 ry 0 rz -180 deg; joints [-145.566, -76.447, -32.214, 64.981, 38.609, -59.152]
  MoveL 9166 to (228.87, 164, 125.68) mm, rotated rx 180 ry 0 rz -180 deg; joints [-145.566, -76.447, -32.214, 64.981, 38.609, -59.152]
  Call Extruder(666.70613)
  MoveL 9167 to (228.64, 164.04, 125.68) mm, rotated rx 180 ry 0 rz -180 deg; joints [-145.551, -76.417, -32.275, 64.959, 38.635, -59.117]
  MoveL 9168 to (228.64, 164.04, 125.68) mm, rotated rx 180 ry 0 rz -180 deg; joints [-145.551, -76.417, -32.275, 64.959, 38.635, -59.117]
  Call Extruder(666.84310)
  MoveL 9169 to (228.4, 164.09, 125.68) mm, rotated rx -180 ry 0 rz 180 deg; joints [-145.535, -76.383, -32.342, 64.934, 38.663, -59.079]
  MoveL 9170 to (228.4, 164.09, 125.68) mm, rotated rx -180 ry 0 rz 180 deg; joints [-145.535, -76.383, -32.342, 64.934, 38.663, -59.079]
  Call Extruder(666.97947)
  MoveL 9171 to (228.15, 164.14, 125.68) mm, rotated rx 180 ry 0 rz 180 deg; joints [-145.518, -76.349, -32.41, 64.909, 38.692, -59.04]
  MoveL 9172 to (228.15, 164.14, 125.68) mm, rotated rx 180 ry 0 rz 180 deg; joints [-145.518, -76.349, -32.41, 64.909, 38.692, -59.04]
  Call Extruder(667.11523)
  MoveL 9173 to (227.9, 164.19, 125.68) mm, rotated rx 180 ry 0 rz 180 deg; joints [-145.502, -76.315, -32.477, 64.885, 38.72, -59.002]
  MoveL 9174 to (227.9, 164.19, 125.68) mm, rotated rx 180 ry 0 rz 180 deg; joints [-145.502, -76.315, -32.477, 64.885, 38.72, -59.002]
  Call Extruder(667.25038)
  MoveL 9175 to (227.65, 164.24, 125.68) mm, rotated rx -180 ry 0 rz 180 deg; joints [-145.485, -76.282, -32.545, 64.86, 38.749, -58.964]
  MoveL 9176 to (227.65, 164.24, 125.68) mm, rotated rx -180 ry 0 rz 180 deg; joints [-145.485, -76.282, -32.545, 64.86, 38.749, -58.964]
  Call Extruder(667.38491)
  MoveL 9177 to (227.4, 164.29, 125.68) mm, rotated rx -180 ry 0 rz 180 deg; joints [-145.469, -76.248, -32.611, 64.836, 38.777, -58.926]
  MoveL 9178 to (227.4, 164.29, 125.68) mm, rotated rx -180 ry 0 rz 180 deg; joints [-145.469, -76.248, -32.611, 64.836, 38.777, -58.926]
  Call Extruder(667.51884)
  MoveL 9179 to (227.15, 164.34, 125.68) mm, rotated rx 180 ry 0 rz 180 deg; joints [-145.453, -76.215, -32.678, 64.812, 38.805, -58.888]
  MoveL 9180 to (227.15, 164.34, 125.68) mm, rotated rx 180 ry 0 rz 180 deg; joints [-145.453, -76.215, -32.678, 64.812, 38.805, -58.888]
  Call Extruder(667.66670)
  MoveL 9181 to (226.87, 164.39, 125.68) mm, rotated rx -180 ry 0 rz -180 deg; joints [-145.435, -76.177, -32.754, 64.784, 38.837, -58.845]
  MoveL 9182 to (226.87, 164.39, 125.68) mm, rotated rx -180 ry 0 rz -180 deg; joints [-145.435, -76.177, -32.754, 64.784, 38.837, -58.845]
  Call Extruder(667.82844)
  MoveL 9183 to (226.57, 164.44, 125.68) mm, rotated rx 180 ry 0 rz 180 deg; joints [-145.415, -76.135, -32.839, 64.753, 38.871, -58.797]
  MoveL 9184 to (226.57, 164.44, 125.68) mm, rotated rx 180 ry 0 rz 180 deg; joints [-145.415, -76.135, -32.839, 64.753, 38.871, -58.797]
  Call Extruder(667.98945)
  MoveL 9185 to (226.26, 164.49, 125.68) mm, rotated rx -180 ry 0 rz -180 deg; joints [-145.396, -76.093, -32.923, 64.721, 38.906, -58.748]
  MoveL 9186 to (226.26, 164.49, 125.68) mm, rotated rx -180 ry 0 rz -180 deg; joints [-145.396, -76.093, -32.923, 64.721, 38.906, -58.748]
  Call Extruder(668.14974)
  MoveL 9187 to (225.96, 164.54, 125.68) mm, rotated rx 180 ry 0 rz 180 deg; joints [-145.377, -76.051, -33.007, 64.69, 38.94, -58.7]
  MoveL 9188 to (225.96, 164.54, 125.68) mm, rotated rx 180 ry 0 rz 180 deg; joints [-145.377, -76.051, -33.007, 64.69, 38.94, -58.7]
  Call Extruder(668.30929)
  MoveL 9189 to (225.65, 164.58, 125.68) mm, rotated rx 180 ry 0 rz -180 deg; joints [-145.357, -76.009, -33.091, 64.659, 38.975, -58.652]
  MoveL 9190 to (225.65, 164.58, 125.68) mm, rotated rx 180 ry 0 rz -180 deg; joints [-145.357, -76.009, -33.091, 64.659, 38.975, -58.652]
  Call Extruder(668.46812)
  MoveL 9191 to (225.34, 164.63, 125.68) mm, rotated rx 180 ry 0 rz 180 deg; joints [-145.338, -75.967, -33.175, 64.628, 39.009, -58.604]
  MoveL 9192 to (225.34, 164.63, 125.68) mm, rotated rx 180 ry 0 rz 180 deg; joints [-145.338, -75.967, -33.175, 64.628, 39.009, -58.604]
  Call Extruder(668.64679)
  MoveL 9193 to (225, 164.68, 125.68) mm, rotated rx -180 ry 0 rz 180 deg; joints [-145.317, -75.919, -33.271, 64.592, 39.048, -58.549]
  MoveL 9194 to (225, 164.68, 125.68) mm, rotated rx -180 ry 0 rz 180 deg; joints [-145.317, -75.919, -33.271, 64.592, 39.048, -58.549]
  Call Extruder(668.84523)
  MoveL 9195 to (224.61, 164.72, 125.68) mm, rotated rx 180 ry 0 rz -180 deg; joints [-145.293, -75.864, -33.38, 64.551, 39.092, -58.486]
  MoveL 9196 to (224.61, 164.72, 125.68) mm, rotated rx 180 ry 0 rz -180 deg; joints [-145.293, -75.864, -33.38, 64.551, 39.092, -58.486]
  Call Extruder(669.04281)
  MoveL 9197 to (224.22, 164.77, 125.68) mm, rotated rx -180 ry 0 rz 180 deg; joints [-145.27, -75.81, -33.489, 64.51, 39.135, -58.423]
  MoveL 9198 to (224.22, 164.77, 125.68) mm, rotated rx -180 ry 0 rz 180 deg; joints [-145.27, -75.81, -33.489, 64.51, 39.135, -58.423]
  Call Extruder(669.23952)
  MoveL 9199 to (223.83, 164.82, 125.68) mm, rotated rx -180 ry 0 rz 180 deg; joints [-145.246, -75.756, -33.597, 64.469, 39.178, -58.36]
  MoveL 9200 to (223.83, 164.82, 125.68) mm, rotated rx -180 ry 0 rz 180 deg; joints [-145.246, -75.756, -33.597, 64.469, 39.178, -58.36]
  Call Extruder(669.43535)
  MoveL 9201 to (223.45, 164.86, 125.68) mm, rotated rx -180 ry 0 rz 180 deg; joints [-145.223, -75.702, -33.706, 64.429, 39.222, -58.298]
  MoveL 9202 to (223.45, 164.86, 125.68) mm, rotated rx -180 ry 0 rz 180 deg; joints [-145.223, -75.702, -33.706, 64.429, 39.222, -58.298]
  Call Extruder(669.73071)
  MoveL 9203 to (222.86, 164.91, 125.68) mm, rotated rx 180 ry 0 rz 180 deg; joints [-145.189, -75.618, -33.874, 64.364, 39.287, -58.199]
  MoveL 9204 to (222.86, 164.91, 125.68) mm, rotated rx 180 ry 0 rz 180 deg; joints [-145.189, -75.618, -33.874, 64.364, 39.287, -58.199]
  Call Extruder(670.02474)
  MoveL 9205 to (222.27, 164.95, 125.68) mm, rotated rx -180 ry 0 rz -180 deg; joints [-145.155, -75.534, -34.043, 64.299, 39.353, -58.101]
  MoveL 9206 to (222.27, 164.95, 125.68) mm, rotated rx -180 ry 0 rz -180 deg; joints [-145.155, -75.534, -34.043, 64.299, 39.353, -58.101]
  Call Extruder(670.31744)
  MoveL 9207 to (221.68, 165, 125.68) mm, rotated rx 180 ry 0 rz 180 deg; joints [-145.121, -75.451, -34.21, 64.236, 39.418, -58.004]
  MoveL 9208 to (221.68, 165, 125.68) mm, rotated rx 180 ry 0 rz 180 deg; joints [-145.121, -75.451, -34.21, 64.236, 39.418, -58.004]
  Call Extruder(670.89088)
  MoveL 9209 to (220.52, 165.05, 125.68) mm, rotated rx 180 ry 0 rz 180 deg; joints [-145.056, -75.282, -34.548, 64.104, 39.546, -57.805]
  MoveL 9210 to (220.52, 165.05, 125.68) mm, rotated rx 180 ry 0 rz 180 deg; joints [-145.056, -75.282, -34.548, 64.104, 39.546, -57.805]
  Call Extruder(671.60489)
  MoveL 9211 to (219.06, 165.09, 125.68) mm, rotated rx -180 ry 0 rz 180 deg; joints [-144.977, -75.071, -34.971, 63.939, 39.706, -57.557]
  Call Extruder(788.45163)
  MoveL 9212 to (-19.06, 165.09, 125.68) mm, rotated rx -180 ry 0 rz 180 deg; joints [-127.434, -54.085, -79.256, 62.282, 63.763, -40.078]
  Call Extruder(788.88023)
  MoveL 9213 to (-19.94, 165.07, 125.68) mm, rotated rx 180 ry 0 rz 180 deg; joints [-127.348, -54.037, -79.365, 62.33, 63.847, -40.05]
  MoveL 9214 to (-19.94, 165.07, 125.68) mm, rotated rx 180 ry 0 rz 180 deg; joints [-127.348, -54.037, -79.365, 62.33, 63.847, -40.05]
  Call Extruder(789.45369)
  MoveL 9215 to (-21.1, 165.02, 125.68) mm, rotated rx 180 ry 0 rz 180 deg; joints [-127.235, -53.972, -79.513, 62.391, 63.959, -40.011]
  MoveL 9216 to (-21.1, 165.02, 125.68) mm, rotated rx 180 ry 0 rz 180 deg; joints [-127.235, -53.972, -79.513, 62.391, 63.959, -40.011]
  Call Extruder(789.88798)
  MoveL 9217 to (-21.97, 164.98, 125.68) mm, rotated rx -180 ry 0 rz 180 deg; joints [-127.15, -53.923, -79.626, 62.436, 64.043, -39.98]
  MoveL 9218 to (-21.97, 164.98, 125.68) mm, rotated rx -180 ry 0 rz 180 deg; joints [-127.15, -53.923, -79.626, 62.436, 64.043, -39.98]
  Call Extruder(790.18201)
  MoveL 9219 to (-22.56, 164.93, 125.68) mm, rotated rx 180 ry 0 rz -180 deg; joints [-127.093, -53.888, -79.704, 62.465, 64.099, -39.958]
  MoveL 9220 to (-22.56, 164.93, 125.68) mm, rotated rx 180 ry 0 rz -180 deg; joints [-127.093, -53.888, -79.704, 62.465, 64.099, -39.958]
  Call Extruder(790.47737)
  MoveL 9221 to (-23.15, 164.89, 125.68) mm, rotated rx -180 ry 0 rz 180 deg; joints [-127.037, -53.854, -79.782, 62.494, 64.155, -39.936]
  MoveL 9222 to (-23.15, 164.89, 125.68) mm, rotated rx -180 ry 0 rz 180 deg; joints [-127.037, -53.854, -79.782, 62.494, 64.155, -39.936]
  Call Extruder(790.72359)
  MoveL 9223 to (-23.64, 164.84, 125.68) mm, rotated rx 180 ry 0 rz -180 deg; joints [-126.991, -53.825, -79.848, 62.517, 64.202, -39.917]
  MoveL 9224 to (-23.64, 164.84, 125.68) mm, rotated rx 180 ry 0 rz -180 deg; joints [-126.991, -53.825, -79.848, 62.517, 64.202, -39.917]
  Call Extruder(790.92030)
  MoveL 9225 to (-24.03, 164.79, 125.68) mm, rotated rx 180 ry 0 rz -180 deg; joints [-126.955, -53.801, -79.901, 62.535, 64.239, -39.9]
  MoveL 9226 to (-24.03, 164.79, 125.68) mm, rotated rx 180 ry 0 rz -180 deg; joints [-126.955, -53.801, -79.901, 62.535, 64.239, -39.9]
  Call Extruder(791.11787)
  MoveL 9227 to (-24.42, 164.75, 125.68) mm, rotated rx -180 ry 0 rz 180 deg; joints [-126.919, -53.778, -79.955, 62.552, 64.276, -39.884]
  MoveL 9228 to (-24.42, 164.75, 125.68) mm, rotated rx -180 ry 0 rz 180 deg; joints [-126.919, -53.778, -79.955, 62.552, 64.276, -39.884]
  Call Extruder(791.31631)
  MoveL 9229 to (-24.8, 164.7, 125.68) mm, rotated rx 180 ry 0 rz 180 deg; joints [-126.883, -53.754, -80.009, 62.57, 64.313, -39.868]
  MoveL 9230 to (-24.8, 164.7, 125.68) mm, rotated rx 180 ry 0 rz 180 deg; joints [-126.883, -53.754, -80.009, 62.57, 64.313, -39.868]
  Call Extruder(791.51562)
  MoveL 9231 to (-25.19, 164.66, 125.68) mm, rotated rx -180 ry 0 rz 180 deg; joints [-126.847, -53.731, -80.062, 62.588, 64.349, -39.851]
  MoveL 9232 to (-25.19, 164.66, 125.68) mm, rotated rx -180 ry 0 rz 180 deg; joints [-126.847, -53.731, -80.062, 62.588, 64.349, -39.851]
  Call Extruder(791.67445)
  MoveL 9233 to (-25.5, 164.61, 125.68) mm, rotated rx 180 ry 0 rz -180 deg; joints [-126.82, -53.711, -80.106, 62.601, 64.378, -39.837]
  MoveL 9234 to (-25.5, 164.61, 125.68) mm, rotated rx 180 ry 0 rz -180 deg; joints [-126.82, -53.711, -80.106, 62.601, 64.378, -39.837]
  Call Extruder(791.83401)
  MoveL 9235 to (-25.8, 164.56, 125.68) mm, rotated rx -180 ry 0 rz 180 deg; joints [-126.792, -53.692, -80.15, 62.614, 64.407, -39.823]
  MoveL 9236 to (-25.8, 164.56, 125.68) mm, rotated rx -180 ry 0 rz 180 deg; joints [-126.792, -53.692, -80.15, 62.614, 64.407, -39.823]
  Call Extruder(791.99430)
  MoveL 9237 to (-26.11, 164.51, 125.68) mm, rotated rx 180 ry 0 rz 180 deg; joints [-126.765, -53.673, -80.194, 62.627, 64.436, -39.809]
  MoveL 9238 to (-26.11, 164.51, 125.68) mm, rotated rx 180 ry 0 rz 180 deg; joints [-126.765, -53.673, -80.194, 62.627, 64.436, -39.809]
  Call Extruder(792.15531)
  MoveL 9239 to (-26.41, 164.46, 125.68) mm, rotated rx 180 ry 0 rz 180 deg; joints [-126.737, -53.654, -80.238, 62.64, 64.465, -39.794]
  MoveL 9240 to (-26.41, 164.46, 125.68) mm, rotated rx 180 ry 0 rz 180 deg; joints [-126.737, -53.654, -80.238, 62.64, 64.465, -39.794]
  Call Extruder(792.31706)
  MoveL 9241 to (-26.72, 164.41, 125.68) mm, rotated rx -180 ry 0 rz 180 deg; joints [-126.71, -53.634, -80.282, 62.653, 64.495, -39.78]
  MoveL 9242 to (-26.72, 164.41, 125.68) mm, rotated rx -180 ry 0 rz 180 deg; joints [-126.71, -53.634, -80.282, 62.653, 64.495, -39.78]
  Call Extruder(792.47953)
  MoveL 9243 to (-27.03, 164.36, 125.68) mm, rotated rx -180 ry 0 rz 180 deg; joints [-126.682, -53.615, -80.326, 62.666, 64.523, -39.766]
  MoveL 9244 to (-27.03, 164.36, 125.68) mm, rotated rx -180 ry 0 rz 180 deg; joints [-126.682, -53.615, -80.326, 62.666, 64.523, -39.766]
  Call Extruder(792.61345)
  MoveL 9245 to (-27.27, 164.32, 125.68) mm, rotated rx -180 ry 0 rz 180 deg; joints [-126.66, -53.599, -80.363, 62.676, 64.547, -39.753]
  MoveL 9246 to (-27.27, 164.32, 125.68) mm, rotated rx -180 ry 0 rz 180 deg; joints [-126.66, -53.599, -80.363, 62.676, 64.547, -39.753]
  Call Extruder(792.74799)
  MoveL 9247 to (-27.52, 164.27, 125.68) mm, rotated rx 180 ry 0 rz 180 deg; joints [-126.638, -53.582, -80.401, 62.685, 64.571, -39.741]
  MoveL 9248 to (-27.52, 164.27, 125.68) mm, rotated rx 180 ry 0 rz 180 deg; joints [-126.638, -53.582, -80.401, 62.685, 64.571, -39.741]
  Call Extruder(792.88314)
  MoveL 9249 to (-27.77, 164.22, 125.68) mm, rotated rx -180 ry 0 rz 180 deg; joints [-126.617, -53.566, -80.438, 62.695, 64.594, -39.728]
  MoveL 9250 to (-27.77, 164.22, 125.68) mm, rotated rx -180 ry 0 rz 180 deg; joints [-126.617, -53.566, -80.438, 62.695, 64.594, -39.728]
  Call Extruder(793.01889)
  MoveL 9251 to (-28.02, 164.17, 125.68) mm, rotated rx 180 ry 0 rz 180 deg; joints [-126.595, -53.55, -80.475, 62.705, 64.618, -39.715]
  MoveL 9252 to (-28.02, 164.17, 125.68) mm, rotated rx 180 ry 0 rz 180 deg; joints [-126.595, -53.55, -80.475, 62.705, 64.618, -39.715]
  Call Extruder(793.15526)
  MoveL 9253 to (-28.27, 164.12, 125.68) mm, rotated rx -180 ry 0 rz 180 deg; joints [-126.573, -53.533, -80.513, 62.714, 64.641, -39.703]
  MoveL 9254 to (-28.27, 164.12, 125.68) mm, rotated rx -180 ry 0 rz 180 deg; joints [-126.573, -53.533, -80.513, 62.714, 64.641, -39.703]
  Call Extruder(793.24012)
  MoveL 9255 to (-28.42, 164.09, 125.68) mm, rotated rx 180 ry 0 rz 180 deg; joints [-126.559, -53.523, -80.536, 62.721, 64.656, -39.695]
  Set speed (130.0 mm/s)
  MoveL 9256 to (-31.76, 163.31, 125.68) mm, rotated rx 180 ry 0 rz -180 deg; joints [-126.274, -53.299, -81.05, 62.843, 64.97, -39.514]
  MoveL 9257 to (-31.76, 163.31, 135.08) mm, rotated rx 180 ry 0 rz -180 deg; joints [-126.274, -52.065, -81.494, 63.174, 64.612, -40.291]
  Call Extruder(791.24012)
  Set speed (40.0 mm/s)
  MoveL 9258 to (-31.76, 163.31, 135.08) mm, rotated rx 180 ry 0 rz -180 deg; joints [-126.274, -52.065, -81.494, 63.174, 64.612, -40.291]
  Call Extruder(0.00000)
  Set speed (130.0 mm/s)
  MoveL 9259 to (-39.41, 155.44, 135.08) mm, rotated rx 180 ry 0 rz -180 deg; joints [-126.075, -51.124, -83.616, 62.851, 65.276, -39.201]
  Call Extruder(2.00000)
  Set speed (40.0 mm/s)
  MoveL 9260 to (-39.41, 155.44, 135.08) mm, rotated rx 180 ry 0 rz -180 deg; joints [-126.075, -51.124, -83.616, 62.851, 65.276, -39.201]
  Set speed (30.0 mm/s)
  MoveL 9261 to (-39.41, 155.44, 135.08) mm, rotated rx 180 ry 0 rz -180 deg; joints [-126.075, -51.124, -83.616, 62.851, 65.276, -39.201]
  Call Extruder(2.05684)
  MoveL 9262 to (-39.44, 155.34, 135.08) mm, rotated rx 180 ry 0 rz 180 deg; joints [-126.079, -51.116, -83.634, 62.843, 65.278, -39.19]
  MoveL 9263 to (-39.44, 155.34, 135.08) mm, rotated rx 180 ry 0 rz 180 deg; joints [-126.079, -51.116, -83.634, 62.843, 65.278, -39.19]
  Call Extruder(2.17007)
  MoveL 9264 to (-39.5, 155.15, 135.08) mm, rotated rx -180 ry 0 rz 180 deg; joints [-126.087, -51.1, -83.671, 62.828, 65.282, -39.167]
  MoveL 9265 to (-39.5, 155.15, 135.08) mm, rotated rx -180 ry 0 rz 180 deg; joints [-126.087, -51.1, -83.671, 62.828, 65.282, -39.167]
  Call Extruder(2.28286)
  MoveL 9266 to (-39.56, 154.97, 135.08) mm, rotated rx 180 ry 0 rz 180 deg; joints [-126.095, -51.084, -83.707, 62.813, 65.286, -39.144]
  MoveL 9267 to (-39.56, 154.97, 135.08) mm, rotated rx 180 ry 0 rz 180 deg; joints [-126.095, -51.084, -83.707, 62.813, 65.286, -39.144]
  Call Extruder(2.39521)
  MoveL 9268 to (-39.62, 154.78, 135.08) mm, rotated rx 180 ry 0 rz -180 deg; joints [-126.103, -51.068, -83.743, 62.797, 65.29, -39.121]
  MoveL 9269 to (-39.62, 154.78, 135.08) mm, rotated rx 180 ry 0 rz -180 deg; joints [-126.103, -51.068, -83.743, 62.797, 65.29, -39.121]
  Call Extruder(2.50711)
  MoveL 9270 to (-39.68, 154.59, 135.08) mm, rotated rx 180 ry 0 rz -180 deg; joints [-126.111, -51.052, -83.78, 62.782, 65.294, -39.099]
  MoveL 9271 to (-39.68, 154.59, 135.08) mm, rotated rx 180 ry 0 rz -180 deg; joints [-126.111, -51.052, -83.78, 62.782, 65.294, -39.099]
  Call Extruder(2.62851)
  MoveL 9272 to (-39.75, 154.38, 135.08) mm, rotated rx 180 ry 0 rz -180 deg; joints [-126.12, -51.035, -83.819, 62.765, 65.299, -39.074]
  MoveL 9273 to (-39.75, 154.38, 135.08) mm, rotated rx 180 ry 0 rz -180 deg; joints [-126.12, -51.035, -83.819, 62.765, 65.299, -39.074]
  Call Extruder(2.75930)
  MoveL 9274 to (-39.81, 154.16, 135.08) mm, rotated rx 180 ry 0 rz 180 deg; joints [-126.131, -51.016, -83.862, 62.747, 65.303, -39.047]
  MoveL 9275 to (-39.81, 154.16, 135.08) mm, rotated rx 180 ry 0 rz 180 deg; joints [-126.131, -51.016, -83.862, 62.747, 65.303, -39.047]
  Call Extruder(2.88953)
  MoveL 9276 to (-39.88, 153.94, 135.08) mm, rotated rx -180 ry 0 rz -180 deg; joints [-126.141, -50.997, -83.904, 62.728, 65.307, -39.02]
  MoveL 9277 to (-39.88, 153.94, 135.08) mm, rotated rx -180 ry 0 rz -180 deg; joints [-126.141, -50.997, -83.904, 62.728, 65.307, -39.02]
  Call Extruder(3.01920)
  MoveL 9278 to (-39.95, 153.71, 135.08) mm, rotated rx 180 ry 0 rz 180 deg; joints [-126.151, -50.978, -83.947, 62.71, 65.312, -38.993]
  MoveL 9279 to (-39.95, 153.71, 135.08) mm, rotated rx 180 ry 0 rz 180 deg; joints [-126.151, -50.978, -83.947, 62.71, 65.312, -38.993]
  Call Extruder(3.14830)
  MoveL 9280 to (-40.02, 153.49, 135.08) mm, rotated rx -180 ry 0 rz 180 deg; joints [-126.161, -50.959, -83.989, 62.691, 65.316, -38.966]
  MoveL 9281 to (-40.02, 153.49, 135.08) mm, rotated rx -180 ry 0 rz 180 deg; joints [-126.161, -50.959, -83.989, 62.691, 65.316, -38.966]
  Call Extruder(3.26338)
  MoveL 9282 to (-40.06, 153.28, 135.08) mm, rotated rx -180 ry 0 rz 180 deg; joints [-126.173, -50.943, -84.026, 62.673, 65.319, -38.942]
  MoveL 9283 to (-40.06, 153.28, 135.08) mm, rotated rx -180 ry 0 rz 180 deg; joints [-126.173, -50.943, -84.026, 62.673, 65.319, -38.942]
  Call Extruder(3.37800)
  MoveL 9284 to (-40.11, 153.08, 135.08) mm, rotated rx -180 ry 0 rz 180 deg; joints [-126.184, -50.927, -84.063, 62.655, 65.321, -38.917]
  MoveL 9285 to (-40.11, 153.08, 135.08) mm, rotated rx -180 ry 0 rz 180 deg; joints [-126.184, -50.927, -84.063, 62.655, 65.321, -38.917]
  Call Extruder(3.49217)
  MoveL 9286 to (-40.15, 152.88, 135.08) mm, rotated rx -180 ry 0 rz 180 deg; joints [-126.195, -50.911, -84.1, 62.637, 65.324, -38.893]
  MoveL 9287 to (-40.15, 152.88, 135.08) mm, rotated rx -180 ry 0 rz 180 deg; joints [-126.195, -50.911, -84.1, 62.637, 65.324, -38.893]
  Call Extruder(3.60589)
  MoveL 9288 to (-40.2, 152.67, 135.08) mm, rotated rx 180 ry 0 rz 180 deg; joints [-126.206, -50.895, -84.137, 62.619, 65.326, -38.869]
  MoveL 9289 to (-40.2, 152.67, 135.08) mm, rotated rx 180 ry 0 rz 180 deg; joints [-126.206, -50.895, -84.137, 62.619, 65.326, -38.869]
  Call Extruder(3.70891)
  MoveL 9290 to (-40.23, 152.49, 135.08) mm, rotated rx 180 ry 0 rz 180 deg; joints [-126.217, -50.88, -84.17, 62.602, 65.328, -38.847]
  MoveL 9291 to (-40.23, 152.49, 135.08) mm, rotated rx 180 ry 0 rz 180 deg; joints [-126.217, -50.88, -84.17, 62.602, 65.328, -38.847]
  Call Extruder(3.80140)
  MoveL 9292 to (-40.27, 152.32, 135.08) mm, rotated rx 180 ry 0 rz 180 deg; joints [-126.226, -50.867, -84.2, 62.587, 65.33, -38.827]
  Set speed (130.0 mm/s)
  MoveL 9293 to (-40.27, 152.32, 135.08) mm, rotated rx 180 ry 0 rz 180 deg; joints [-126.226, -50.867, -84.2, 62.587, 65.33, -38.827]
  Set speed (30.0 mm/s)
  MoveL 9294 to (-40.27, 152.32, 135.08) mm, rotated rx 180 ry 0 rz 180 deg; joints [-126.226, -50.867, -84.2, 62.587, 65.33, -38.827]
  Call Extruder(3.93780)
  MoveL 9295 to (-40.32, 152.07, 135.08) mm, rotated rx -180 ry 0 rz -180 deg; joints [-126.241, -50.847, -84.244, 62.565, 65.332, -38.798]
  MoveL 9296 to (-40.32, 152.07, 135.08) mm, rotated rx -180 ry 0 rz -180 deg; joints [-126.241, -50.847, -84.244, 62.565, 65.332, -38.798]
  Call Extruder(4.07360)
  MoveL 9297 to (-40.37, 151.82, 135.08) mm, rotated rx -180 ry 0 rz 180 deg; joints [-126.255, -50.828, -84.289, 62.543, 65.335, -38.769]
  MoveL 9298 to (-40.37, 151.82, 135.08) mm, rotated rx -180 ry 0 rz 180 deg; joints [-126.255, -50.828, -84.289, 62.543, 65.335, -38.769]
  Call Extruder(4.20879)
  MoveL 9299 to (-40.42, 151.57, 135.08) mm, rotated rx 180 ry 0 rz 180 deg; joints [-126.269, -50.808, -84.333, 62.52, 65.337, -38.739]
  MoveL 9300 to (-40.42, 151.57, 135.08) mm, rotated rx 180 ry 0 rz 180 deg; joints [-126.269, -50.808, -84.333, 62.52, 65.337, -38.739]
  Call Extruder(4.34337)
  MoveL 9301 to (-40.47, 151.32, 135.08) mm, rotated rx 180 ry 0 rz 180 deg; joints [-126.283, -50.789, -84.377, 62.498, 65.34, -38.71]
  MoveL 9302 to (-40.47, 151.32, 135.08) mm, rotated rx 180 ry 0 rz 180 deg; joints [-126.283, -50.789, -84.377, 62.498, 65.34, -38.71]
  Call Extruder(4.47734)
  MoveL 9303 to (-40.52, 151.07, 135.08) mm, rotated rx 180 ry 0 rz 180 deg; joints [-126.298, -50.77, -84.421, 62.476, 65.342, -38.681]
  MoveL 9304 to (-40.52, 151.07, 135.08) mm, rotated rx 180 ry 0 rz 180 deg; joints [-126.298, -50.77, -84.421, 62.476, 65.342, -38.681]
  Call Extruder(4.61071)
  MoveL 9305 to (-40.57, 150.82, 135.08) mm, rotated rx -180 ry 0 rz 180 deg; joints [-126.312, -50.75, -84.465, 62.453, 65.345, -38.651]
  MoveL 9306 to (-40.57, 150.82, 135.08) mm, rotated rx -180 ry 0 rz 180 deg; joints [-126.312, -50.75, -84.465, 62.453, 65.345, -38.651]
  Call Extruder(4.77280)
  MoveL 9307 to (-40.61, 150.52, 135.08) mm, rotated rx 180 ry 0 rz -180 deg; joints [-126.331, -50.727, -84.518, 62.425, 65.347, -38.616]
